        function block Node_F_VN_MaxElementElementwise_TcVnVector3_REAL [ST]: FB_init, Clone, OnExecute, PreExecutionCheck
        function block Node_F_VN_MaxElementElementwise_TcVnVector3_SINT [ST]: FB_init, Clone, OnExecute, PreExecutionCheck
        function block Node_F_VN_MaxElementElementwise_TcVnVector3_UINT [ST]: FB_init, Clone, OnExecute, PreExecutionCheck
        function block Node_F_VN_MaxElementElementwise_TcVnVector3_USINT [ST]: FB_init, Clone, OnExecute, PreExecutionCheck
        function block Node_F_VN_MaxElementElementwise_TcVnVector4_DINT [ST]: FB_init, Clone, OnExecute, PreExecutionCheck
        function block Node_F_VN_MaxElementElementwise_TcVnVector4_INT [ST]: FB_init, Clone, OnExecute, PreExecutionCheck
        function block Node_F_VN_MaxElementElementwise_TcVnVector4_LREAL [ST]: FB_init, Clone, OnExecute, PreExecutionCheck
        function block Node_F_VN_MaxElementElementwise_TcVnVector4_REAL [ST]: FB_init, Clone, OnExecute, PreExecutionCheck
        function block Node_F_VN_MaxElementElementwise_TcVnVector4_SINT [ST]: FB_init, Clone, OnExecute, PreExecutionCheck
        function block Node_F_VN_MaxElementElementwise_TcVnVector4_UINT [ST]: FB_init, Clone, OnExecute, PreExecutionCheck
        function block Node_F_VN_MaxElementElementwise_TcVnVector4_USINT [ST]: FB_init, Clone, OnExecute, PreExecutionCheck
        function block Node_F_VN_MaxElementElementwise_UDINT [ST]: FB_init, Clone, OnExecute, PreExecutionCheck
        function block Node_F_VN_MaxElementElementwise_UINT [ST]: FB_init, Clone, OnExecute, PreExecutionCheck
        function block Node_F_VN_MaxElementElementwise_ULINT [ST]: FB_init, Clone, OnExecute, PreExecutionCheck
        function block Node_F_VN_MaxElementElementwise_USINT [ST]: FB_init, Clone, OnExecute, PreExecutionCheck
      MedianElementwise/
        function block Node_F_VN_MedianElementElementwise_DINT [ST]: FB_init, Clone, OnExecute, PreExecutionCheck
        function block Node_F_VN_MedianElementElementwise_INT [ST]: FB_init, Clone, OnExecute, PreExecutionCheck
        function block Node_F_VN_MedianElementElementwise_LREAL [ST]: FB_init, Clone, OnExecute, PreExecutionCheck
        function block Node_F_VN_MedianElementElementwise_REAL [ST]: FB_init, Clone, OnExecute, PreExecutionCheck
        function block Node_F_VN_MedianElementElementwise_SINT [ST]: FB_init, Clone, OnExecute, PreExecutionCheck
        function block Node_F_VN_MedianElementElementwise_TcVnPoint2_DINT [ST]: FB_init, Clone, OnExecute, PreExecutionCheck
        function block Node_F_VN_MedianElementElementwise_TcVnPoint2_LREAL [ST]: FB_init, Clone, OnExecute, PreExecutionCheck
        function block Node_F_VN_MedianElementElementwise_TcVnPoint2_REAL [ST]: FB_init, Clone, OnExecute, PreExecutionCheck
        function block Node_F_VN_MedianElementElementwise_TcVnPoint3_LREAL [ST]: FB_init, Clone, OnExecute, PreExecutionCheck
        function block Node_F_VN_MedianElementElementwise_TcVnPoint3_REAL [ST]: FB_init, Clone, OnExecute, PreExecutionCheck
        function block Node_F_VN_MedianElementElementwise_TcVnVector2_DINT [ST]: FB_init, Clone, OnExecute, PreExecutionCheck
        function block Node_F_VN_MedianElementElementwise_TcVnVector2_INT [ST]: FB_init, Clone, OnExecute, PreExecutionCheck
        function block Node_F_VN_MedianElementElementwise_TcVnVector2_REAL [ST]: FB_init, Clone, OnExecute, PreExecutionCheck
        function block Node_F_VN_MedianElementElementwise_TcVnVector2_SINT [ST]: FB_init, Clone, OnExecute, PreExecutionCheck
        function block Node_F_VN_MedianElementElementwise_TcVnVector2_UINT [ST]: FB_init, Clone, OnExecute, PreExecutionCheck
        function block Node_F_VN_MedianElementElementwise_TcVnVector2_USINT [ST]: FB_init, Clone, OnExecute, PreExecutionCheck
        function block Node_F_VN_MedianElementElementwise_TcVnVector3_INT [ST]: FB_init, Clone, OnExecute, PreExecutionCheck
        function block Node_F_VN_MedianElementElementwise_TcVnVector3_REAL [ST]: FB_init, Clone, OnExecute, PreExecutionCheck
        function block Node_F_VN_MedianElementElementwise_TcVnVector3_SINT [ST]: FB_init, Clone, OnExecute, PreExecutionCheck
        function block Node_F_VN_MedianElementElementwise_TcVnVector3_UINT [ST]: FB_init, Clone, OnExecute, PreExecutionCheck
        function block Node_F_VN_MedianElementElementwise_TcVnVector3_USINT [ST]: FB_init, Clone, OnExecute, PreExecutionCheck
        function block Node_F_VN_MedianElementElementwise_TcVnVector4_DINT [ST]: FB_init, Clone, OnExecute, PreExecutionCheck
        function block Node_F_VN_MedianElementElementwise_TcVnVector4_INT [ST]: FB_init, Clone, OnExecute, PreExecutionCheck
        function block Node_F_VN_MedianElementElementwise_TcVnVector4_LREAL [ST]: FB_init, Clone, OnExecute, PreExecutionCheck
        function block Node_F_VN_MedianElementElementwise_TcVnVector4_REAL [ST]: FB_init, Clone, OnExecute, PreExecutionCheck
        function block Node_F_VN_MedianElementElementwise_TcVnVector4_SINT [ST]: FB_init, Clone, OnExecute, PreExecutionCheck
        function block Node_F_VN_MedianElementElementwise_TcVnVector4_UINT [ST]: FB_init, Clone, OnExecute, PreExecutionCheck
        function block Node_F_VN_MedianElementElementwise_TcVnVector4_USINT [ST]: FB_init, Clone, OnExecute, PreExecutionCheck
        function block Node_F_VN_MedianElementElementwise_UDINT [ST]: FB_init, Clone, OnExecute, PreExecutionCheck
        function block Node_F_VN_MedianElementElementwise_UINT [ST]: FB_init, Clone, OnExecute, PreExecutionCheck
        function block Node_F_VN_MedianElementElementwise_ULINT [ST]: FB_init, Clone, OnExecute, PreExecutionCheck
        function block Node_F_VN_MedianElementElementwise_USINT [ST]: FB_init, Clone, OnExecute, PreExecutionCheck
      MinElementwise/
        function block Node_F_VN_MinElementElementwise_DINT [ST]: FB_init, Clone, OnExecute, PreExecutionCheck
        function block Node_F_VN_MinElementElementwise_INT [ST]: FB_init, Clone, OnExecute, PreExecutionCheck
        function block Node_F_VN_MinElementElementwise_LREAL [ST]: FB_init, Clone, OnExecute, PreExecutionCheck
        function block Node_F_VN_MinElementElementwise_REAL [ST]: FB_init, Clone, OnExecute, PreExecutionCheck
        function block Node_F_VN_MinElementElementwise_SINT [ST]: FB_init, Clone, OnExecute, PreExecutionCheck
        function block Node_F_VN_MinElementElementwise_TcVnPoint2_DINT [ST]: FB_init, Clone, OnExecute, PreExecutionCheck
        function block Node_F_VN_MinElementElementwise_TcVnPoint2_LREAL [ST]: FB_init, Clone, OnExecute, PreExecutionCheck
        function block Node_F_VN_MinElementElementwise_TcVnPoint2_REAL [ST]: FB_init, Clone, OnExecute, PreExecutionCheck
        function block Node_F_VN_MinElementElementwise_TcVnPoint3_LREAL [ST]: FB_init, Clone, OnExecute, PreExecutionCheck
        function block Node_F_VN_MinElementElementwise_TcVnPoint3_REAL [ST]: FB_init, Clone, OnExecute, PreExecutionCheck
        function block Node_F_VN_MinElementElementwise_TcVnVector2_DINT [ST]: FB_init, Clone, OnExecute, PreExecutionCheck
        function block Node_F_VN_MinElementElementwise_TcVnVector2_INT [ST]: FB_init, Clone, OnExecute, PreExecutionCheck
        function block Node_F_VN_MinElementElementwise_TcVnVector2_REAL [ST]: FB_init, Clone, OnExecute, PreExecutionCheck
        function block Node_F_VN_MinElementElementwise_TcVnVector2_SINT [ST]: FB_init, Clone, OnExecute, PreExecutionCheck
        function block Node_F_VN_MinElementElementwise_TcVnVector2_UINT [ST]: FB_init, Clone, OnExecute, PreExecutionCheck
        function block Node_F_VN_MinElementElementwise_TcVnVector2_USINT [ST]: FB_init, Clone, OnExecute, PreExecutionCheck
        function block Node_F_VN_MinElementElementwise_TcVnVector3_INT [ST]: FB_init, Clone, OnExecute, PreExecutionCheck
        function block Node_F_VN_MinElementElementwise_TcVnVector3_REAL [ST]: FB_init, Clone, OnExecute, PreExecutionCheck
        function block Node_F_VN_MinElementElementwise_TcVnVector3_SINT [ST]: FB_init, Clone, OnExecute, PreExecutionCheck
        function block Node_F_VN_MinElementElementwise_TcVnVector3_UINT [ST]: FB_init, Clone, OnExecute, PreExecutionCheck
        function block Node_F_VN_MinElementElementwise_TcVnVector3_USINT [ST]: FB_init, Clone, OnExecute, PreExecutionCheck
        function block Node_F_VN_MinElementElementwise_TcVnVector4_DINT [ST]: FB_init, Clone, OnExecute, PreExecutionCheck
        function block Node_F_VN_MinElementElementwise_TcVnVector4_INT [ST]: FB_init, Clone, OnExecute, PreExecutionCheck
        function block Node_F_VN_MinElementElementwise_TcVnVector4_LREAL [ST]: FB_init, Clone, OnExecute, PreExecutionCheck
        function block Node_F_VN_MinElementElementwise_TcVnVector4_REAL [ST]: FB_init, Clone, OnExecute, PreExecutionCheck
        function block Node_F_VN_MinElementElementwise_TcVnVector4_SINT [ST]: FB_init, Clone, OnExecute, PreExecutionCheck
        function block Node_F_VN_MinElementElementwise_TcVnVector4_UINT [ST]: FB_init, Clone, OnExecute, PreExecutionCheck
        function block Node_F_VN_MinElementElementwise_TcVnVector4_USINT [ST]: FB_init, Clone, OnExecute, PreExecutionCheck
        function block Node_F_VN_MinElementElementwise_UDINT [ST]: FB_init, Clone, OnExecute, PreExecutionCheck
        function block Node_F_VN_MinElementElementwise_UINT [ST]: FB_init, Clone, OnExecute, PreExecutionCheck
        function block Node_F_VN_MinElementElementwise_ULINT [ST]: FB_init, Clone, OnExecute, PreExecutionCheck
        function block Node_F_VN_MinElementElementwise_USINT [ST]: FB_init, Clone, OnExecute, PreExecutionCheck
      function block Node_F_VN_ContainerAverage [ST]: FB_init, Clone, OnExecute, PreExecutionCheck
      function block Node_F_VN_ContainerAverageElementwise2 [ST]: FB_init, Clone, OnExecute, PreExecutionCheck
      function block Node_F_VN_ContainerAverageElementwise3 [ST]: FB_init, Clone, OnExecute, PreExecutionCheck
      function block Node_F_VN_ContainerAverageElementwise4 [ST]: FB_init, Clone, OnExecute, PreExecutionCheck
      function block Node_F_VN_ContainerAverageVariance [ST]: FB_init, Clone, OnExecute, PreExecutionCheck
      function block Node_F_VN_ContainerAverageVarianceElementwise2 [ST]: FB_init, Clone, OnExecute, PreExecutionCheck
      function block Node_F_VN_ContainerAverageVarianceElementwise3 [ST]: FB_init, Clone, OnExecute, PreExecutionCheck
      function block Node_F_VN_ContainerAverageVarianceElementwise4 [ST]: FB_init, Clone, OnExecute, PreExecutionCheck
      function block Node_F_VN_MaxElement [ST]: FB_init, Clone, OnExecute, PreExecutionCheck
      function block Node_F_VN_MedianElement [ST]: FB_init, Clone, OnExecute, PreExecutionCheck
      function block Node_F_VN_MinElement [ST]: FB_init, Clone, OnExecute, PreExecutionCheck
    Contour Analysis/
      function block Node_F_VN_ApproximatePolygon [ST]: FB_init, Clone, OnExecute, PreExecutionCheck
      function block Node_F_VN_CheckIfPointIsInsideContour [ST]: FB_init, Clone, OnExecute, PreExecutionCheck
      function block Node_F_VN_ContourArea [ST]: FB_init, Clone, OnExecute, PreExecutionCheck
      function block Node_F_VN_ContourCenterOfMass [ST]: FB_init, Clone, OnExecute, PreExecutionCheck
      function block Node_F_VN_ContourCircularity [ST]: FB_init, Clone, OnExecute, PreExecutionCheck
      function block Node_F_VN_ContourCircularityExp [ST]: FB_init, Clone, OnExecute, PreExecutionCheck
      function block Node_F_VN_ContourConvexity [ST]: FB_init, Clone, OnExecute, PreExecutionCheck
      function block Node_F_VN_ContourEccentricity [ST]: FB_init, Clone, OnExecute, PreExecutionCheck
      function block Node_F_VN_ContourElongation [ST]: FB_init, Clone, OnExecute, PreExecutionCheck
      function block Node_F_VN_ContourExtremePoint [ST]: FB_init, Clone, OnExecute, PreExecutionCheck
      function block Node_F_VN_ContourInertiaRatio [ST]: FB_init, Clone, OnExecute, PreExecutionCheck
      function block Node_F_VN_ContourMoments [ST]: FB_init, Clone, OnExecute, PreExecutionCheck
      function block Node_F_VN_ContourOrientation [ST]: FB_init, Clone, OnExecute, PreExecutionCheck
      function block Node_F_VN_ContourOrientationExp [ST]: FB_init, Clone, OnExecute, PreExecutionCheck
      function block Node_F_VN_ContourPerimeter [ST]: FB_init, Clone, OnExecute, PreExecutionCheck
      function block Node_F_VN_ContourRoundness [ST]: FB_init, Clone, OnExecute, PreExecutionCheck
      function block Node_F_VN_ConvexHullPoints [ST]: FB_init, Clone, OnExecute, PreExecutionCheck
      function block Node_F_VN_ConvexHullPointsExp [ST]: FB_init, Clone, OnExecute, PreExecutionCheck
      function block Node_F_VN_ConvexityDefects [ST]: FB_init, Clone, OnExecute, PreExecutionCheck
      function block Node_F_VN_EnclosingCircle [ST]: FB_init, Clone, OnExecute, PreExecutionCheck
      function block Node_F_VN_EnclosingRectangle [ST]: FB_init, Clone, OnExecute, PreExecutionCheck
      function block Node_F_VN_EnclosingTriangle [ST]: FB_init, Clone, OnExecute, PreExecutionCheck
      function block Node_F_VN_FitEllipse [ST]: FB_init, Clone, OnExecute, PreExecutionCheck
      function block Node_F_VN_FitLine [ST]: FB_init, Clone, OnExecute, PreExecutionCheck
      function block Node_F_VN_FitLineExp [ST]: FB_init, Clone, OnExecute, PreExecutionCheck
      function block Node_F_VN_MatchContours [ST]: FB_init, Clone, OnExecute, PreExecutionCheck
      function block Node_F_VN_MatchContours1vsN [ST]: FB_init, Clone, OnExecute, PreExecutionCheck
      function block Node_F_VN_MatchContours1vsNExp [ST]: FB_init, Clone, OnExecute, PreExecutionCheck
      function block Node_F_VN_MatchContoursExp [ST]: FB_init, Clone, OnExecute, PreExecutionCheck
      function block Node_F_VN_UprightBoundingRectangle [ST]: FB_init, Clone, OnExecute, PreExecutionCheck
    Control Functions/
    Drawing/
      function block Node_F_VN_DrawArrow [ST]: FB_init, Clone, OnExecute, PreExecutionCheck
      function block Node_F_VN_DrawArrow_TcVnVector4_DINT [ST]: FB_init, Clone, OnExecute, PreExecutionCheck
      function block Node_F_VN_DrawArrowExp [ST]: FB_init, Clone, OnExecute, PreExecutionCheck
      function block Node_F_VN_DrawArrowExp_TcVnVector4_DINT [ST]: FB_init, Clone, OnExecute, PreExecutionCheck
      function block Node_F_VN_DrawCircle [ST]: FB_init, Clone, OnExecute, PreExecutionCheck
      function block Node_F_VN_DrawCircleExp [ST]: FB_init, Clone, OnExecute, PreExecutionCheck
      function block Node_F_VN_DrawCircles [ST]: FB_init, Clone, OnExecute, PreExecutionCheck
      function block Node_F_VN_DrawCirclesExp [ST]: FB_init, Clone, OnExecute, PreExecutionCheck
      function block Node_F_VN_DrawCircularArc [ST]: FB_init, Clone, OnExecute, PreExecutionCheck
      function block Node_F_VN_DrawCircularArcExp [ST]: FB_init, Clone, OnExecute, PreExecutionCheck
      function block Node_F_VN_DrawComponents [ST]: FB_init, Clone, OnExecute, PreExecutionCheck
      function block Node_F_VN_DrawComponentsExp [ST]: FB_init, Clone, OnExecute, PreExecutionCheck
      function block Node_F_VN_DrawContours [ST]: FB_init, Clone, OnExecute, PreExecutionCheck
      function block Node_F_VN_DrawContoursExp [ST]: FB_init, Clone, OnExecute, PreExecutionCheck
      function block Node_F_VN_DrawEllipse [ST]: FB_init, Clone, OnExecute, PreExecutionCheck
      function block Node_F_VN_DrawEllipseExp [ST]: FB_init, Clone, OnExecute, PreExecutionCheck
      function block Node_F_VN_DrawKeypoints [ST]: FB_init, Clone, OnExecute, PreExecutionCheck
      function block Node_F_VN_DrawKeypointsExp [ST]: FB_init, Clone, OnExecute, PreExecutionCheck
      function block Node_F_VN_DrawLine [ST]: FB_init, Clone, OnExecute, PreExecutionCheck
      function block Node_F_VN_DrawLine_TcVnVector4_DINT [ST]: FB_init, Clone, OnExecute, PreExecutionCheck
      function block Node_F_VN_DrawLine_TcVnVector4_LREAL [ST]: FB_init, Clone, OnExecute, PreExecutionCheck
      function block Node_F_VN_DrawLineExp [ST]: FB_init, Clone, OnExecute, PreExecutionCheck
      function block Node_F_VN_DrawLineExp_TcVnVector4_DINT [ST]: FB_init, Clone, OnExecute, PreExecutionCheck
      function block Node_F_VN_DrawLineExp_TcVnVector4_LREAL [ST]: FB_init, Clone, OnExecute, PreExecutionCheck
      function block Node_F_VN_DrawLines [ST]: FB_init, Clone, OnExecute, PreExecutionCheck
      function block Node_F_VN_DrawLinesExp [ST]: FB_init, Clone, OnExecute, PreExecutionCheck
      function block Node_F_VN_DrawMatches [ST]: FB_init, Clone, OnExecute, PreExecutionCheck
      function block Node_F_VN_DrawMatchesExp [ST]: FB_init, Clone, OnExecute, PreExecutionCheck
      function block Node_F_VN_DrawOrientation [ST]: FB_init, Clone, OnExecute, PreExecutionCheck
      function block Node_F_VN_DrawOrientationExp [ST]: FB_init, Clone, OnExecute, PreExecutionCheck
      function block Node_F_VN_DrawPoint [ST]: FB_init, Clone, OnExecute, PreExecutionCheck
      function block Node_F_VN_DrawPointExp [ST]: FB_init, Clone, OnExecute, PreExecutionCheck
      function block Node_F_VN_DrawPoints [ST]: FB_init, Clone, OnExecute, PreExecutionCheck
      function block Node_F_VN_DrawPointsExp [ST]: FB_init, Clone, OnExecute, PreExecutionCheck
      function block Node_F_VN_DrawPolygon [ST]: FB_init, Clone, OnExecute, PreExecutionCheck
      function block Node_F_VN_DrawPolygonExp [ST]: FB_init, Clone, OnExecute, PreExecutionCheck
      function block Node_F_VN_DrawRectangle [ST]: FB_init, Clone, OnExecute, PreExecutionCheck
      function block Node_F_VN_DrawRectangle_TcVnRectangle_DINT [ST]: FB_init, Clone, OnExecute, PreExecutionCheck
      function block Node_F_VN_DrawRectangle_TcVnRectangle_UDINT [ST]: FB_init, Clone, OnExecute, PreExecutionCheck
      function block Node_F_VN_DrawRotatedRectangle [ST]: FB_init, Clone, OnExecute, PreExecutionCheck
      function block Node_F_VN_DrawRotatedRectangleExp [ST]: FB_init, Clone, OnExecute, PreExecutionCheck
      function block Node_F_VN_FillCircle [ST]: FB_init, Clone, OnExecute, PreExecutionCheck
      function block Node_F_VN_FillContours [ST]: FB_init, Clone, OnExecute, PreExecutionCheck
      function block Node_F_VN_FillEllipse [ST]: FB_init, Clone, OnExecute, PreExecutionCheck
      function block Node_F_VN_FillPolygon [ST]: FB_init, Clone, OnExecute, PreExecutionCheck
      function block Node_F_VN_FillRectangle [ST]: FB_init, Clone, OnExecute, PreExecutionCheck
      function block Node_F_VN_FillRotatedRectangle [ST]: FB_init, Clone, OnExecute, PreExecutionCheck
      function block Node_F_VN_PlotIntensityProfile [ST]: FB_init, Clone, OnExecute, PreExecutionCheck
      function block Node_F_VN_PlotIntensityProfileExp [ST]: FB_init, Clone, OnExecute, PreExecutionCheck
      function block Node_F_VN_PutLabel [ST]: FB_init, Clone, OnExecute, PreExecutionCheck
      function block Node_F_VN_PutLabelExp [ST]: FB_init, Clone, OnExecute, PreExecutionCheck
      function block Node_F_VN_PutText [ST]: FB_init, Clone, OnExecute, PreExecutionCheck
      function block Node_F_VN_PutTextExp [ST]: FB_init, Clone, OnExecute, PreExecutionCheck
    Fourier Analysis/
      function block Node_F_VN_CreateBandpassButterworthFilter [ST]: FB_init, Clone, OnExecute, PreExecutionCheck
      function block Node_F_VN_CreateBandpassGaussianFilter [ST]: FB_init, Clone, OnExecute, PreExecutionCheck
      function block Node_F_VN_CreateBandrejectButterworthFilter [ST]: FB_init, Clone, OnExecute, PreExecutionCheck
      function block Node_F_VN_CreateBandrejectGaussianFilter [ST]: FB_init, Clone, OnExecute, PreExecutionCheck
      function block Node_F_VN_CreateHighpassButterworthFilter [ST]: FB_init, Clone, OnExecute, PreExecutionCheck
      function block Node_F_VN_CreateHighpassGaussianFilter [ST]: FB_init, Clone, OnExecute, PreExecutionCheck
      function block Node_F_VN_CreateLowpassButterworthFilter [ST]: FB_init, Clone, OnExecute, PreExecutionCheck
      function block Node_F_VN_CreateLowpassGaussianFilter [ST]: FB_init, Clone, OnExecute, PreExecutionCheck
      function block Node_F_VN_Dft [ST]: FB_init, Clone, OnExecute, PreExecutionCheck
      function block Node_F_VN_InverseDft [ST]: FB_init, Clone, OnExecute, PreExecutionCheck
      function block Node_F_VN_OptimalDftSize [ST]: FB_init, Clone, OnExecute, PreExecutionCheck
    Geometric and Coord Transform/
      Calibration/
        function block Node_F_VN_CalibrateCamera [ST]: FB_init, Clone, OnExecute, PreExecutionCheck
        function block Node_F_VN_CalibrateCameraPlanar [ST]: FB_init, Clone, OnExecute, PreExecutionCheck
        function block Node_F_VN_CompensateLensDistortion [ST]: FB_init, Clone, OnExecute, PreExecutionCheck
        function block Node_F_VN_CompensateLensDistortionExp1 [ST]: FB_init, Clone, OnExecute, PreExecutionCheck
        function block Node_F_VN_CompensateLensDistortionExp2 [ST]: FB_init, Clone, OnExecute, PreExecutionCheck
        function block Node_F_VN_CompensateLensDistortionForPoints [ST]: FB_init, Clone, OnExecute, PreExecutionCheck
        function block Node_F_VN_CompensateLensDistortionForPointsExp1 [ST]: FB_init, Clone, OnExecute, PreExecutionCheck
        function block Node_F_VN_CompensateLensDistortionForPointsExp2 [ST]: FB_init, Clone, OnExecute, PreExecutionCheck
        function block Node_F_VN_DetectPatternPoints [ST]: FB_init, Clone, OnExecute, PreExecutionCheck
        function block Node_F_VN_GenerateCalibrationPatternReferencePoints [ST]: FB_init, Clone, OnExecute, PreExecutionCheck
        function block Node_F_VN_SolvePnP [ST]: FB_init, Clone, OnExecute, PreExecutionCheck
        function block Node_F_VN_SolvePnPExp [ST]: FB_init, Clone, OnExecute, PreExecutionCheck
        function block Node_F_VN_SortDetectedPatternPoints [ST]: FB_init, Clone, OnExecute, PreExecutionCheck
      function block Node_F_VN_AlignRotatedImageRegion [ST]: FB_init, Clone, OnExecute, PreExecutionCheck
      function block Node_F_VN_AlignRotatedImageRegionExp [ST]: FB_init, Clone, OnExecute, PreExecutionCheck
      function block Node_F_VN_ApplyRotationToAffineTransformation [ST]: FB_init, Clone, OnExecute, PreExecutionCheck
      function block Node_F_VN_ApplyRotationToAffineTransformationExp [ST]: FB_init, Clone, OnExecute, PreExecutionCheck
      function block Node_F_VN_ApplyScalingToAffineTransformation [ST]: FB_init, Clone, OnExecute, PreExecutionCheck
      function block Node_F_VN_ApplyScalingToAffineTransformationExp [ST]: FB_init, Clone, OnExecute, PreExecutionCheck
      function block Node_F_VN_ApplyTranslationToAffineTransformation [ST]: FB_init, Clone, OnExecute, PreExecutionCheck
      function block Node_F_VN_ApplyTranslationToAffineTransformationExp [ST]: FB_init, Clone, OnExecute, PreExecutionCheck
      function block Node_F_VN_ApplyYAxisInversionToAffineTransformation [ST]: FB_init, Clone, OnExecute, PreExecutionCheck
      function block Node_F_VN_ApplyYAxisInversionToAffineTransformationExp [ST]: FB_init, Clone, OnExecute, PreExecutionCheck
      function block Node_F_VN_ConvertCartesianToPolarAngleImage [ST]: FB_init, Clone, OnExecute, PreExecutionCheck
      function block Node_F_VN_ConvertCartesianToPolarAngleImageExp [ST]: FB_init, Clone, OnExecute, PreExecutionCheck
      function block Node_F_VN_ConvertCartesianToPolarAngles [ST]: FB_init, Clone, OnExecute, PreExecutionCheck
      function block Node_F_VN_ConvertCartesianToPolarAnglesExp [ST]: FB_init, Clone, OnExecute, PreExecutionCheck
      function block Node_F_VN_ConvertCartesianToPolarImages [ST]: FB_init, Clone, OnExecute, PreExecutionCheck
      function block Node_F_VN_ConvertCartesianToPolarImagesExp [ST]: FB_init, Clone, OnExecute, PreExecutionCheck
      function block Node_F_VN_ConvertCartesianToPolarMagnitudeImage [ST]: FB_init, Clone, OnExecute, PreExecutionCheck
      function block Node_F_VN_ConvertCartesianToPolarMagnitudes [ST]: FB_init, Clone, OnExecute, PreExecutionCheck
      function block Node_F_VN_ConvertCartesianToPolarPoints [ST]: FB_init, Clone, OnExecute, PreExecutionCheck
      function block Node_F_VN_ConvertCartesianToPolarPointsExp [ST]: FB_init, Clone, OnExecute, PreExecutionCheck
      function block Node_F_VN_ConvertMaps [ST]: FB_init, Clone, OnExecute, PreExecutionCheck
      function block Node_F_VN_ConvertPolarToCartesianImages [ST]: FB_init, Clone, OnExecute, PreExecutionCheck
      function block Node_F_VN_ConvertPolarToCartesianImagesExp [ST]: FB_init, Clone, OnExecute, PreExecutionCheck
      function block Node_F_VN_ConvertPolarToCartesianPoints [ST]: FB_init, Clone, OnExecute, PreExecutionCheck
      function block Node_F_VN_ConvertPolarToCartesianPointsExp [ST]: FB_init, Clone, OnExecute, PreExecutionCheck
      function block Node_F_VN_DecomposeAffineTransformation [ST]: FB_init, Clone, OnExecute, PreExecutionCheck
      function block Node_F_VN_DecomposeAffineTransformationExp [ST]: FB_init, Clone, OnExecute, PreExecutionCheck
      function block Node_F_VN_FlipImage [ST]: FB_init, Clone, OnExecute, PreExecutionCheck
      function block Node_F_VN_GenerateAffineTransformationUnitMatrix2D [ST]: FB_init, Clone, OnExecute, PreExecutionCheck
      function block Node_F_VN_GetAffineTransformation [ST]: FB_init, Clone, OnExecute, PreExecutionCheck
      function block Node_F_VN_GetAffineTransformation2D [ST]: FB_init, Clone, OnExecute, PreExecutionCheck
      function block Node_F_VN_GetPerspectiveTransformation [ST]: FB_init, Clone, OnExecute, PreExecutionCheck
      function block Node_F_VN_Homography [ST]: FB_init, Clone, OnExecute, PreExecutionCheck
      function block Node_F_VN_HomographyExp [ST]: FB_init, Clone, OnExecute, PreExecutionCheck
      function block Node_F_VN_InvertAffineTransformation [ST]: FB_init, Clone, OnExecute, PreExecutionCheck
      function block Node_F_VN_PerspectiveTransformation [ST]: FB_init, Clone, OnExecute, PreExecutionCheck
      function block Node_F_VN_PyramidDown [ST]: FB_init, Clone, OnExecute, PreExecutionCheck
      function block Node_F_VN_PyramidUp [ST]: FB_init, Clone, OnExecute, PreExecutionCheck
      function block Node_F_VN_RemapImage [ST]: FB_init, Clone, OnExecute, PreExecutionCheck
      function block Node_F_VN_RemapImageExp [ST]: FB_init, Clone, OnExecute, PreExecutionCheck
      function block Node_F_VN_RemapImageToLogPolarSpace [ST]: FB_init, Clone, OnExecute, PreExecutionCheck
      function block Node_F_VN_RemapImageToLogPolarSpaceExp [ST]: FB_init, Clone, OnExecute, PreExecutionCheck
      function block Node_F_VN_RemapImageToLogPolarSpaceExp2 [ST]: FB_init, Clone, OnExecute, PreExecutionCheck
      function block Node_F_VN_RemapImageToPolarSpace [ST]: FB_init, Clone, OnExecute, PreExecutionCheck
      function block Node_F_VN_RemapImageToPolarSpaceExp [ST]: FB_init, Clone, OnExecute, PreExecutionCheck
      function block Node_F_VN_RemapImageToPolarSpaceExp2 [ST]: FB_init, Clone, OnExecute, PreExecutionCheck
      function block Node_F_VN_ResizeImage [ST]: FB_init, Clone, OnExecute, PreExecutionCheck
      function block Node_F_VN_ResizeImageExp [ST]: FB_init, Clone, OnExecute, PreExecutionCheck
      function block Node_F_VN_ResizeRegion_TcVnRectangle_DINT [ST]: FB_init, Clone, OnExecute, PreExecutionCheck
      function block Node_F_VN_RotateImage [ST]: FB_init, Clone, OnExecute, PreExecutionCheck
      function block Node_F_VN_RotateImageExp [ST]: FB_init, Clone, OnExecute, PreExecutionCheck
      function block Node_F_VN_RotateImageExp2 [ST]: FB_init, Clone, OnExecute, PreExecutionCheck
      function block Node_F_VN_WarpAffine [ST]: FB_init, Clone, OnExecute, PreExecutionCheck
      function block Node_F_VN_WarpAffine_Container [ST]: FB_init, Clone, OnExecute, PreExecutionCheck
      function block Node_F_VN_WarpAffine_Point [ST]: FB_init, Clone, OnExecute, PreExecutionCheck
      function block Node_F_VN_WarpAffine_Rectangle [ST]: FB_init, Clone, OnExecute, PreExecutionCheck
      function block Node_F_VN_WarpAffineExp [ST]: FB_init, Clone, OnExecute, PreExecutionCheck
      function block Node_F_VN_WarpPerspective [ST]: FB_init, Clone, OnExecute, PreExecutionCheck
      function block Node_F_VN_WarpPerspective_Container [ST]: FB_init, Clone, OnExecute, PreExecutionCheck
      function block Node_F_VN_WarpPerspective_Point [ST]: FB_init, Clone, OnExecute, PreExecutionCheck
      function block Node_F_VN_WarpPerspective_Rectangle [ST]: FB_init, Clone, OnExecute, PreExecutionCheck
      function block Node_F_VN_WarpPerspectiveExp [ST]: FB_init, Clone, OnExecute, PreExecutionCheck
    Helpers/
      function block Node_Mux10Way_ITcVnImage [ST]: FB_init, Clone, OnExecute
    Image Analysis/
      Object Detection/
        function block Node_F_VN_DetectBlobs [ST]: FB_init, Clone, OnExecute, PreExecutionCheck
        function block Node_F_VN_DetectBlobsExp [ST]: FB_init, Clone, OnExecute, PreExecutionCheck
        function block Node_F_VN_FindContourHierarchyExp [ST]: FB_init, Clone, OnExecute, PreExecutionCheck
        function block Node_F_VN_FindContours [ST]: FB_init, Clone, OnExecute, PreExecutionCheck
        function block Node_F_VN_FindContoursExp [ST]: FB_init, Clone, OnExecute, PreExecutionCheck
        function block Node_F_VN_FindRois [ST]: FB_init, Clone, OnExecute, PreExecutionCheck
        function block Node_F_VN_FindTemplateWalsh [ST]: FB_init, Clone, OnExecute, PreExecutionCheck
        function block Node_F_VN_FindTemplateWalsh_AngleRange [ST]: FB_init, Clone, OnExecute, PreExecutionCheck
        function block Node_F_VN_FindTemplateWalshExp [ST]: FB_init, Clone, OnExecute, PreExecutionCheck
        function block Node_F_VN_FindTemplateWalshExp_AngleRange [ST]: FB_init, Clone, OnExecute, PreExecutionCheck
        function block Node_F_VN_HoughCircles [ST]: FB_init, Clone, OnExecute, PreExecutionCheck
        function block Node_F_VN_HoughCirclesExp [ST]: FB_init, Clone, OnExecute, PreExecutionCheck
        function block Node_F_VN_HoughLines [ST]: FB_init, Clone, OnExecute, PreExecutionCheck
        function block Node_F_VN_HoughLinesP [ST]: FB_init, Clone, OnExecute, PreExecutionCheck
        function block Node_F_VN_HoughLinesPExp [ST]: FB_init, Clone, OnExecute, PreExecutionCheck
        function block Node_F_VN_MatchImageHuMoments [ST]: FB_init, Clone, OnExecute, PreExecutionCheck
        function block Node_F_VN_MatchTemplate [ST]: FB_init, Clone, OnExecute, PreExecutionCheck
        function block Node_F_VN_MatchTemplateAndEvaluate [ST]: FB_init, Clone, OnExecute, PreExecutionCheck
        function block Node_F_VN_MatchTemplateAndEvaluateExp [ST]: FB_init, Clone, OnExecute, PreExecutionCheck
        function block Node_F_VN_MatchTemplateExp [ST]: FB_init, Clone, OnExecute, PreExecutionCheck
        function block Node_F_VN_MatchTemplateWalsh [ST]: FB_init, Clone, OnExecute, PreExecutionCheck
        function block Node_F_VN_MatchTemplateWalshExp [ST]: FB_init, Clone, OnExecute, PreExecutionCheck
        function block Node_F_VN_MergeRegions [ST]: FB_init, Clone, OnExecute, PreExecutionCheck
        function block Node_F_VN_SalientFeatures [ST]: FB_init, Clone, OnExecute, PreExecutionCheck
      function block Node_F_VN_CannyEdgeDetection [ST]: FB_init, Clone, OnExecute, PreExecutionCheck
      function block Node_F_VN_CannyEdgeDetectionExp [ST]: FB_init, Clone, OnExecute, PreExecutionCheck
      function block Node_F_VN_ConnectedComponents [ST]: FB_init, Clone, OnExecute, PreExecutionCheck
      function block Node_F_VN_ConnectedComponentsExp [ST]: FB_init, Clone, OnExecute, PreExecutionCheck
      function block Node_F_VN_ConnectedComponentsWithStats [ST]: FB_init, Clone, OnExecute, PreExecutionCheck
      function block Node_F_VN_ConnectedComponentsWithStatsExp [ST]: FB_init, Clone, OnExecute, PreExecutionCheck
      function block Node_F_VN_CountNonZeroPixels [ST]: FB_init, Clone, OnExecute, PreExecutionCheck
      function block Node_F_VN_DistanceTransformation [ST]: FB_init, Clone, OnExecute, PreExecutionCheck
      function block Node_F_VN_DistanceTransformationExp [ST]: FB_init, Clone, OnExecute, PreExecutionCheck
      function block Node_F_VN_GetConnectedComponent [ST]: FB_init, Clone, OnExecute, PreExecutionCheck
      function block Node_F_VN_GetConnectedComponentExp [ST]: FB_init, Clone, OnExecute, PreExecutionCheck
      function block Node_F_VN_ImageAbsoluteAverage [ST]: FB_init, Clone, OnExecute, PreExecutionCheck
      function block Node_F_VN_ImageAverage [ST]: FB_init, Clone, OnExecute, PreExecutionCheck
      function block Node_F_VN_ImageAverageExp [ST]: FB_init, Clone, OnExecute, PreExecutionCheck
      function block Node_F_VN_ImageAverageStdDev [ST]: FB_init, Clone, OnExecute, PreExecutionCheck
      function block Node_F_VN_ImageAverageStdDevExp [ST]: FB_init, Clone, OnExecute, PreExecutionCheck
      function block Node_F_VN_ImageCenterOfMass [ST]: FB_init, Clone, OnExecute, PreExecutionCheck
      function block Node_F_VN_ImageCenterOfMassExp [ST]: FB_init, Clone, OnExecute, PreExecutionCheck
      function block Node_F_VN_ImageMedian [ST]: FB_init, Clone, OnExecute, PreExecutionCheck
      function block Node_F_VN_ImageMedianExp [ST]: FB_init, Clone, OnExecute, PreExecutionCheck
      function block Node_F_VN_ImageMoments [ST]: FB_init, Clone, OnExecute, PreExecutionCheck
      function block Node_F_VN_MaxPixelValue [ST]: FB_init, Clone, OnExecute, PreExecutionCheck
      function block Node_F_VN_MaxPixelValueExp [ST]: FB_init, Clone, OnExecute, PreExecutionCheck
      function block Node_F_VN_MinPixelValue [ST]: FB_init, Clone, OnExecute, PreExecutionCheck
      function block Node_F_VN_MinPixelValueExp [ST]: FB_init, Clone, OnExecute, PreExecutionCheck
      function block Node_F_VN_RegionOrientation [ST]: FB_init, Clone, OnExecute, PreExecutionCheck
      function block Node_F_VN_RegionOrientationExp [ST]: FB_init, Clone, OnExecute, PreExecutionCheck
      function block Node_F_VN_UprightInnerRectangle [ST]: FB_init, Clone, OnExecute, PreExecutionCheck
      function block Node_F_VN_UprightInnerRectangleExp [ST]: FB_init, Clone, OnExecute, PreExecutionCheck
    Image Color and Contrast Processing/
      function block Node_F_VN_ApplyColorMap [ST]: FB_init, Clone, OnExecute, PreExecutionCheck
      function block Node_F_VN_Clahe [ST]: FB_init, Clone, OnExecute, PreExecutionCheck
      function block Node_F_VN_ClaheExp [ST]: FB_init, Clone, OnExecute, PreExecutionCheck
      function block Node_F_VN_ConvertColorSpace [ST]: FB_init, Clone, OnExecute, PreExecutionCheck
      function block Node_F_VN_GenerateColorMap [ST]: FB_init, Clone, OnExecute, PreExecutionCheck
      function block Node_F_VN_GenerateCustomColorMap [ST]: FB_init, Clone, OnExecute, PreExecutionCheck
      function block Node_F_VN_Histogram [ST]: FB_init, Clone, OnExecute, PreExecutionCheck
      function block Node_F_VN_HistogramEqualization [ST]: FB_init, Clone, OnExecute, PreExecutionCheck
      function block Node_F_VN_HistogramEqualizationExp [ST]: FB_init, Clone, OnExecute, PreExecutionCheck
      function block Node_F_VN_HistogramExp [ST]: FB_init, Clone, OnExecute, PreExecutionCheck
      function block Node_F_VN_InvertImageColor [ST]: FB_init, Clone, OnExecute, PreExecutionCheck
      function block Node_F_VN_InvertImageColorExp [ST]: FB_init, Clone, OnExecute, PreExecutionCheck
      function block Node_F_VN_NormalizeImage [ST]: FB_init, Clone, OnExecute, PreExecutionCheck
      function block Node_F_VN_NormalizeImageExp [ST]: FB_init, Clone, OnExecute, PreExecutionCheck
      function block Node_F_VN_NormalizeImageForDisplay [ST]: FB_init, Clone, OnExecute, PreExecutionCheck
      function block Node_F_VN_ReferenceColorSimilarity_TcVnVector3_LREAL [ST]: FB_init, Clone, OnExecute, PreExecutionCheck
      function block Node_F_VN_ReferenceColorSimilarityExp_TcVnVector3_LREAL [ST]: FB_init, Clone, OnExecute, PreExecutionCheck
      function block Node_F_VN_WhiteBalance [ST]: FB_init, Clone, OnExecute, PreExecutionCheck
    Image Filtering/
      function block Node_F_VN_BilateralFilter [ST]: FB_init, Clone, OnExecute, PreExecutionCheck
      function block Node_F_VN_BilateralFilterExp [ST]: FB_init, Clone, OnExecute, PreExecutionCheck
      function block Node_F_VN_BoxFilter [ST]: FB_init, Clone, OnExecute, PreExecutionCheck
      function block Node_F_VN_BoxFilterExp [ST]: FB_init, Clone, OnExecute, PreExecutionCheck
      function block Node_F_VN_BrightBorderObjects [ST]: FB_init, Clone, OnExecute, PreExecutionCheck
      function block Node_F_VN_CreateStructuringElement [ST]: FB_init, Clone, OnExecute, PreExecutionCheck
      function block Node_F_VN_DarkBorderObjects [ST]: FB_init, Clone, OnExecute, PreExecutionCheck
      function block Node_F_VN_FillHoles [ST]: FB_init, Clone, OnExecute, PreExecutionCheck
      function block Node_F_VN_GaussianFilter [ST]: FB_init, Clone, OnExecute, PreExecutionCheck
      function block Node_F_VN_GaussianFilterExp [ST]: FB_init, Clone, OnExecute, PreExecutionCheck
      function block Node_F_VN_LaplacianFilter [ST]: FB_init, Clone, OnExecute, PreExecutionCheck
      function block Node_F_VN_LaplacianFilterExp [ST]: FB_init, Clone, OnExecute, PreExecutionCheck
      function block Node_F_VN_LocalMaxima [ST]: FB_init, Clone, OnExecute, PreExecutionCheck
      function block Node_F_VN_LocalMinima [ST]: FB_init, Clone, OnExecute, PreExecutionCheck
      function block Node_F_VN_MedianFilter [ST]: FB_init, Clone, OnExecute, PreExecutionCheck
      function block Node_F_VN_MorphologicalOperator [ST]: FB_init, Clone, OnExecute, PreExecutionCheck
      function block Node_F_VN_RemoveLocalMaxima [ST]: FB_init, Clone, OnExecute, PreExecutionCheck
      function block Node_F_VN_RemoveLocalMinima [ST]: FB_init, Clone, OnExecute, PreExecutionCheck
      function block Node_F_VN_ScharrFilter [ST]: FB_init, Clone, OnExecute, PreExecutionCheck
      function block Node_F_VN_ScharrFilterExp [ST]: FB_init, Clone, OnExecute, PreExecutionCheck
      function block Node_F_VN_SobelFilter [ST]: FB_init, Clone, OnExecute, PreExecutionCheck
      function block Node_F_VN_SobelFilterExp [ST]: FB_init, Clone, OnExecute, PreExecutionCheck
      function block Node_F_VN_VarianceFilter [ST]: FB_init, Clone, OnExecute, PreExecutionCheck
      function block Node_F_VN_VarianceFilterExp [ST]: FB_init, Clone, OnExecute, PreExecutionCheck
    Image Segmentation/
      function block Node_F_VN_AdaptiveThreshold [ST]: FB_init, Clone, OnExecute, PreExecutionCheck
      function block Node_F_VN_AdaptiveThresholdExp [ST]: FB_init, Clone, OnExecute, PreExecutionCheck
      function block Node_F_VN_CheckColorRange [ST]: FB_init, Clone, OnExecute, PreExecutionCheck
      function block Node_F_VN_DoubleThreshold [ST]: FB_init, Clone, OnExecute, PreExecutionCheck
      function block Node_F_VN_SauvolaThreshold [ST]: FB_init, Clone, OnExecute, PreExecutionCheck
      function block Node_F_VN_Threshold [ST]: FB_init, Clone, OnExecute, PreExecutionCheck
      function block Node_F_VN_WatershedSegmentationExp [ST]: FB_init, Clone, OnExecute, PreExecutionCheck
    Keypoint Features/
      function block Node_F_VN_FilterGoodMatches [ST]: FB_init, Clone, OnExecute, PreExecutionCheck
      function block Node_F_VN_FindReferenceKeyPointsInImage [ST]: FB_init, Clone, OnExecute, PreExecutionCheck
      function block Node_F_VN_FindReferenceKeyPointsInImageAKAZE [ST]: FB_init, Clone, OnExecute, PreExecutionCheck
      function block Node_F_VN_FindReferenceKeyPointsInImageAKAZEExp [ST]: FB_init, Clone, OnExecute, PreExecutionCheck
      function block Node_F_VN_FindReferenceKeyPointsInImageBRISK [ST]: FB_init, Clone, OnExecute, PreExecutionCheck
      function block Node_F_VN_FindReferenceKeyPointsInImageBRISKExp [ST]: FB_init, Clone, OnExecute, PreExecutionCheck
      function block Node_F_VN_FindReferenceKeyPointsInImageExp [ST]: FB_init, Clone, OnExecute, PreExecutionCheck
      function block Node_F_VN_FindReferenceKeyPointsInImageORB [ST]: FB_init, Clone, OnExecute, PreExecutionCheck
      function block Node_F_VN_FindReferenceKeyPointsInImageORBExp [ST]: FB_init, Clone, OnExecute, PreExecutionCheck
      function block Node_F_VN_GetMatchCoordinates [ST]: FB_init, Clone, OnExecute, PreExecutionCheck
      function block Node_F_VN_KeyPointsAGAST [ST]: FB_init, Clone, OnExecute, PreExecutionCheck
      function block Node_F_VN_KeyPointsAGASTExp [ST]: FB_init, Clone, OnExecute, PreExecutionCheck
      function block Node_F_VN_KeyPointsAndDescriptorsAKAZE [ST]: FB_init, Clone, OnExecute, PreExecutionCheck
      function block Node_F_VN_KeyPointsAndDescriptorsAKAZEExp [ST]: FB_init, Clone, OnExecute, PreExecutionCheck
      function block Node_F_VN_KeyPointsAndDescriptorsBRISK [ST]: FB_init, Clone, OnExecute, PreExecutionCheck
      function block Node_F_VN_KeyPointsAndDescriptorsBRISKExp [ST]: FB_init, Clone, OnExecute, PreExecutionCheck
      function block Node_F_VN_KeyPointsAndDescriptorsKAZE [ST]: FB_init, Clone, OnExecute, PreExecutionCheck
      function block Node_F_VN_KeyPointsAndDescriptorsKAZEExp [ST]: FB_init, Clone, OnExecute, PreExecutionCheck
      function block Node_F_VN_KeyPointsAndDescriptorsORB [ST]: FB_init, Clone, OnExecute, PreExecutionCheck
      function block Node_F_VN_KeyPointsAndDescriptorsORBExp [ST]: FB_init, Clone, OnExecute, PreExecutionCheck
      function block Node_F_VN_KeyPointsFAST [ST]: FB_init, Clone, OnExecute, PreExecutionCheck
      function block Node_F_VN_KeyPointsFASTExp [ST]: FB_init, Clone, OnExecute, PreExecutionCheck
      function block Node_F_VN_KeyPointsGFTT [ST]: FB_init, Clone, OnExecute, PreExecutionCheck
      function block Node_F_VN_KeyPointsGFTTExp [ST]: FB_init, Clone, OnExecute, PreExecutionCheck
      function block Node_F_VN_KeyPointsMSER [ST]: FB_init, Clone, OnExecute, PreExecutionCheck
      function block Node_F_VN_KeyPointsMSERExp [ST]: FB_init, Clone, OnExecute, PreExecutionCheck
      function block Node_F_VN_KeyPointsSB [ST]: FB_init, Clone, OnExecute, PreExecutionCheck
      function block Node_F_VN_KeyPointsSBExp [ST]: FB_init, Clone, OnExecute, PreExecutionCheck
      function block Node_F_VN_MatchDescriptorsBF [ST]: FB_init, Clone, OnExecute, PreExecutionCheck
      function block Node_F_VN_MatchDescriptorsBFExp [ST]: FB_init, Clone, OnExecute, PreExecutionCheck
      function block Node_F_VN_MatchDescriptorsFlannLsh [ST]: FB_init, Clone, OnExecute, PreExecutionCheck
      function block Node_F_VN_MatchDescriptorsFlannLshExp [ST]: FB_init, Clone, OnExecute, PreExecutionCheck
      function block Node_F_VN_MatchDescriptorsKnnBF [ST]: FB_init, Clone, OnExecute, PreExecutionCheck
      function block Node_F_VN_MatchDescriptorsKnnBFExp [ST]: FB_init, Clone, OnExecute, PreExecutionCheck
      function block Node_F_VN_MatchDescriptorsKnnFlannLsh [ST]: FB_init, Clone, OnExecute, PreExecutionCheck
      function block Node_F_VN_MatchDescriptorsKnnFlannLshExp [ST]: FB_init, Clone, OnExecute, PreExecutionCheck
      function block Node_F_VN_RegionsMSER [ST]: FB_init, Clone, OnExecute, PreExecutionCheck
      function block Node_F_VN_RegionsMSERExp [ST]: FB_init, Clone, OnExecute, PreExecutionCheck
    Machine Learning/
    Measurement/
      function block Node_F_VN_AdjustSearchWindowOrientationToLinearEdge [ST]: FB_init, Clone, OnExecute, PreExecutionCheck
      function block Node_F_VN_ClosestPointsBF [ST]: FB_init, Clone, OnExecute, PreExecutionCheck
      function block Node_F_VN_LocateAxisAlignedEdges [ST]: FB_init, Clone, OnExecute, PreExecutionCheck
      function block Node_F_VN_LocateAxisAlignedEdgesExp [ST]: FB_init, Clone, OnExecute, PreExecutionCheck
      function block Node_F_VN_LocateCircularArc [ST]: FB_init, Clone, OnExecute, PreExecutionCheck
      function block Node_F_VN_LocateCircularArcExp [ST]: FB_init, Clone, OnExecute, PreExecutionCheck
      function block Node_F_VN_LocateCircularArcExp2 [ST]: FB_init, Clone, OnExecute, PreExecutionCheck
      function block Node_F_VN_LocateEdge [ST]: FB_init, Clone, OnExecute, PreExecutionCheck
      function block Node_F_VN_LocateEdgeExp [ST]: FB_init, Clone, OnExecute, PreExecutionCheck
      function block Node_F_VN_LocateEdgeExp2 [ST]: FB_init, Clone, OnExecute, PreExecutionCheck
      function block Node_F_VN_LocateEdges [ST]: FB_init, Clone, OnExecute, PreExecutionCheck
      function block Node_F_VN_LocateEdgesExp [ST]: FB_init, Clone, OnExecute, PreExecutionCheck
      function block Node_F_VN_LocateEdgesExp2 [ST]: FB_init, Clone, OnExecute, PreExecutionCheck
      function block Node_F_VN_LocateEllipse [ST]: FB_init, Clone, OnExecute, PreExecutionCheck
      function block Node_F_VN_LocateEllipseExp [ST]: FB_init, Clone, OnExecute, PreExecutionCheck
      function block Node_F_VN_LocateEllipseExp2 [ST]: FB_init, Clone, OnExecute, PreExecutionCheck
      function block Node_F_VN_MeasureAngleBetweenEdges [ST]: FB_init, Clone, OnExecute, PreExecutionCheck
      function block Node_F_VN_MeasureAngleBetweenEdgesExp [ST]: FB_init, Clone, OnExecute, PreExecutionCheck
      function block Node_F_VN_MeasureAngleBetweenEdgesExp2 [ST]: FB_init, Clone, OnExecute, PreExecutionCheck
      function block Node_F_VN_MeasureEdgeDistance [ST]: FB_init, Clone, OnExecute, PreExecutionCheck
      function block Node_F_VN_MeasureEdgeDistanceExp [ST]: FB_init, Clone, OnExecute, PreExecutionCheck
      function block Node_F_VN_MeasureEdgeDistanceExp2 [ST]: FB_init, Clone, OnExecute, PreExecutionCheck
      function block Node_F_VN_MeasureMinEdgeDistance [ST]: FB_init, Clone, OnExecute, PreExecutionCheck
      function block Node_F_VN_MeasureMinEdgeDistanceExp [ST]: FB_init, Clone, OnExecute, PreExecutionCheck
      function block Node_F_VN_MeasureMinEdgeDistanceExp2 [ST]: FB_init, Clone, OnExecute, PreExecutionCheck
    Miscellaneous/
      function block Node_F_VN_CheckFunctionInitialization [ST]: FB_init, Clone, OnExecute, PreExecutionCheck
      function block Node_F_VN_ClipLineToBoundary [ST]: FB_init, Clone, OnExecute, PreExecutionCheck
      function block Node_F_VN_ClipLineToBoundary_ITcVnImage [ST]: FB_init, Clone, OnExecute, PreExecutionCheck
      function block Node_F_VN_ClipLineToBoundary_TcVnRectangle_DINT [ST]: FB_init, Clone, OnExecute, PreExecutionCheck
      function block Node_F_VN_DeinitializeFunction [ST]: FB_init, Clone, OnExecute, PreExecutionCheck
      function block Node_F_VN_HuMomentInvariants [ST]: FB_init, Clone, OnExecute, PreExecutionCheck
      function block Node_F_VN_InvertMatrix3x3 [ST]: FB_init, Clone, OnExecute, PreExecutionCheck
      function block Node_F_VN_LineIntersectionPoint [ST]: FB_init, Clone, OnExecute, PreExecutionCheck
      function block Node_F_VN_LineIntersectionPointAndAngle [ST]: FB_init, Clone, OnExecute, PreExecutionCheck
      function block Node_F_VN_OrthogonalVector_TcVnVector2_DINT [ST]: FB_init, Clone, OnExecute, PreExecutionCheck
      function block Node_F_VN_OrthogonalVector_TcVnVector2_LREAL [ST]: FB_init, Clone, OnExecute, PreExecutionCheck
      function block Node_F_VN_OrthogonalVector_TcVnVector2_REAL [ST]: FB_init, Clone, OnExecute, PreExecutionCheck
      function block Node_F_VN_PointToLineDistance_TcVnPoint2_DINT [ST]: FB_init, Clone, OnExecute, PreExecutionCheck
      function block Node_F_VN_PointToLineDistance_TcVnPoint2_LREAL [ST]: FB_init, Clone, OnExecute, PreExecutionCheck
      function block Node_F_VN_PointToLineDistance_TcVnPoint2_REAL [ST]: FB_init, Clone, OnExecute, PreExecutionCheck
      function block Node_F_VN_PointToPointDirection_TcVnPoint2_DINT [ST]: FB_init, Clone, OnExecute, PreExecutionCheck
      function block Node_F_VN_PointToPointDirection_TcVnPoint2_LREAL [ST]: FB_init, Clone, OnExecute, PreExecutionCheck
      function block Node_F_VN_PointToPointDirection_TcVnPoint2_REAL [ST]: FB_init, Clone, OnExecute, PreExecutionCheck
      function block Node_F_VN_PointToPointDistance_TcVnPoint2_DINT [ST]: FB_init, Clone, OnExecute, PreExecutionCheck
      function block Node_F_VN_PointToPointDistance_TcVnPoint2_LREAL [ST]: FB_init, Clone, OnExecute, PreExecutionCheck
      function block Node_F_VN_PointToPointDistance_TcVnPoint2_REAL [ST]: FB_init, Clone, OnExecute, PreExecutionCheck
      function block Node_F_VN_RotatedRectangleCorners [ST]: FB_init, Clone, OnExecute, PreExecutionCheck
      function block Node_F_VN_RotatedRectangleIntersection [ST]: FB_init, Clone, OnExecute, PreExecutionCheck
    Neural Network/
      function block Node_F_VN_Reduce [ST]: FB_init, Clone, OnExecute, PreExecutionCheck
      function block Node_F_VN_ReduceArg [ST]: FB_init, Clone, OnExecute, PreExecutionCheck
      function block Node_F_VN_Sigmoid [ST]: FB_init, Clone, OnExecute, PreExecutionCheck
      function block Node_F_VN_SigmoidExp [ST]: FB_init, Clone, OnExecute, PreExecutionCheck
      function block Node_F_VN_SoftMax [ST]: FB_init, Clone, OnExecute, PreExecutionCheck
    OCR/
      function block Node_F_VN_OCR [ST]: FB_init, Clone, OnExecute, PreExecutionCheck
      function block Node_F_VN_OCRExp [ST]: FB_init, Clone, OnExecute, PreExecutionCheck
    Polarization/
      function block Node_F_VN_AngleAndDegreeOfLinearPolarization [ST]: FB_init, Clone, OnExecute, PreExecutionCheck
      function block Node_F_VN_DemosaicPolarizedImage [ST]: FB_init, Clone, OnExecute, PreExecutionCheck
      function block Node_F_VN_PolarizedImageGlareReduction [ST]: FB_init, Clone, OnExecute, PreExecutionCheck
    Texture Analysis/
      function block Node_F_VN_Granulometry [ST]: FB_init, Clone, OnExecute, PreExecutionCheck
      function block Node_F_VN_HaralickFeatures [ST]: FB_init, Clone, OnExecute, PreExecutionCheck
    VisionNode/
      function block VisionHardwareNode [ST]: Execute, PreExecutionCheck
      function block VisionNode [ST]: Execute, PreExecutionCheck
    function block VisionNodePack [ST]: RegisterWithNodeFactory
  global variables GVL_COLOURS
  function block VisionPack [ST]: Register
*)

// GVL_COLOURS
{attribute 'qualified_only'}
VAR_GLOBAL
    RGBA_BLACK    : TcVnVector4_LREAL := [0, 0, 0, 255];
    RGBA_RED      : TcVnVector4_LREAL := [255, 0, 0, 255];
    RGBA_YELLOW   : TcVnVector4_LREAL := [255, 255, 0, 255];
    RGBA_GREEN    : TcVnVector4_LREAL := [0, 255, 0, 255];
    RGBA_CYAN     : TcVnVector4_LREAL := [0, 255, 255, 255];
    RGBA_BLUE     : TcVnVector4_LREAL := [0, 0, 255, 255];
    RGBA_MAGENTA  : TcVnVector4_LREAL := [255, 0, 255, 255];
    RGBA_WHITE    : TcVnVector4_LREAL := [255, 255, 255, 255];
    RGBA_RANDOM   : TcVnVector4_LREAL := [-1, -1, -1, -1];
END_VAR

// Datatypes/Aliases/_GVCP_REGISTER_ADDRESS
{attribute 'linkalways'} 
{attribute 'no_explicit_call' := 'This FB is a CLASS and must be accessed using methods or properties'}
{attribute 'enable_dynamic_creation'}
FUNCTION_BLOCK _GVCP_REGISTER_ADDRESS EXTENDS AliasDatatypeBase
VAR
	localData : GVCP_REGISTER_ADDRESS;
	activeData : REFERENCE TO GVCP_REGISTER_ADDRESS REF= localData;
	aliasBaseDatatype : _UDINT(0);
END_VAR

METHOD PROTECTED SetBaseDatatypeReference
VAR_INPUT
END_VAR
aliasBaseDatatype.MakeReferenceTo(activeData);
END_METHOD

PROPERTY PUBLIC Address : PVOID
GET
Address := ADR(activeData);
END_GET
END_PROPERTY

METHOD PUBLIC ClearReference
VAR_INPUT
END_VAR
activeData REF= localData;
SetBaseDatatypeReference();
END_METHOD

PROPERTY PUBLIC Size : UDINT
GET
Size := SIZEOF(activeData);
END_GET
END_PROPERTY

METHOD FB_init : BOOL
VAR_INPUT
	bInitRetains : BOOL; // if TRUE, the retain variables are initialized (warm start / cold start)
	bInCopyCode : BOOL;  // if TRUE, the instance afterwards gets moved into the copy code (online change)
	InitialValue : GVCP_REGISTER_ADDRESS; // if possible, not all values can be initialized
END_VAR
localData := InitialValue;
SetBaseDatatypeReference();
AddBaseDatatype(aliasBaseDatatype);
END_METHOD

METHOD PUBLIC Clone : I_Datatype
VAR
    pClone : POINTER TO _GVCP_REGISTER_ADDRESS;
END_VAR
pClone := __NEW(_GVCP_REGISTER_ADDRESS(InitialValue := Value));
Clone := pClone^;
END_METHOD

PROPERTY PUBLIC Identifier : T_MAXSTRING
GET
Identifier := 'GVCP_REGISTER_ADDRESS';
END_GET
END_PROPERTY

METHOD PUBLIC MakeReferenceTo
VAR_INPUT
	ReferenceTarget : REFERENCE TO GVCP_REGISTER_ADDRESS;
END_VAR
activeData REF= ReferenceTarget;
SetBaseDatatypeReference();
END_METHOD

METHOD TryMakeReferenceTo : BOOL
VAR_INPUT
	Target : I_Datatype;
END_VAR
VAR
	pTargetData : POINTER TO GVCP_REGISTER_ADDRESS;
END_VAR
IF NOT IsEquivalentTo(Target) THEN
	RETURN;
END_IF

pTargetData := Target.Address;
activeData REF= pTargetData^;
SetBaseDatatypeReference();
TryMakeReferenceTo := TRUE;
END_METHOD

PROPERTY PUBLIC Value : REFERENCE TO GVCP_REGISTER_ADDRESS
GET
Value REF= activeData;
END_GET
END_PROPERTY

END_FUNCTION_BLOCK

// Datatypes/Aliases/_GVCP_REGISTER_VALUE
{attribute 'linkalways'}
{attribute 'no_explicit_call' := 'This FB is a CLASS and must be accessed using methods or properties'}
{attribute 'enable_dynamic_creation'}
FUNCTION_BLOCK _GVCP_REGISTER_VALUE EXTENDS AliasDatatypeBase
VAR
	localData : GVCP_REGISTER_VALUE;
	activeData : REFERENCE TO GVCP_REGISTER_VALUE REF= localData;
	aliasBaseDatatype : _UDINT(0);
END_VAR

METHOD PROTECTED SetBaseDatatypeReference
VAR_INPUT
END_VAR
aliasBaseDatatype.MakeReferenceTo(activeData);
END_METHOD

PROPERTY PUBLIC Address : PVOID
GET
Address := ADR(activeData);
END_GET
END_PROPERTY

METHOD PUBLIC ClearReference
VAR_INPUT
END_VAR
activeData REF= localData;
SetBaseDatatypeReference();
END_METHOD

PROPERTY PUBLIC Size : UDINT
GET
Size := SIZEOF(activeData);
END_GET
END_PROPERTY

METHOD FB_init : BOOL
VAR_INPUT
	bInitRetains : BOOL; // if TRUE, the retain variables are initialized (warm start / cold start)
	bInCopyCode : BOOL;  // if TRUE, the instance afterwards gets moved into the copy code (online change)
	InitialValue : GVCP_REGISTER_VALUE := 0;
END_VAR
localData := InitialValue;
SetBaseDatatypeReference();
AddBaseDatatype(aliasBaseDatatype);
END_METHOD

METHOD PUBLIC Clone : I_Datatype
VAR
    pClone : POINTER TO _GVCP_REGISTER_VALUE;
END_VAR
pClone := __NEW(_GVCP_REGISTER_VALUE(InitialValue := Value));
IF pClone = 0 THEN
    RETURN;
END_IF
pClone^.TryCopyFrom(THIS^);
Clone := pClone^;
END_METHOD

PROPERTY PUBLIC Identifier : T_MAXSTRING
GET
Identifier := 'GVCP_REGISTER_VALUE';
END_GET
END_PROPERTY

METHOD PUBLIC MakeReferenceTo
VAR_INPUT
	ReferenceTarget : REFERENCE TO GVCP_REGISTER_VALUE;
END_VAR
activeData REF= ReferenceTarget;
SetBaseDatatypeReference();
END_METHOD

METHOD TryMakeReferenceTo : BOOL
VAR_INPUT
	Target : I_Datatype;
END_VAR
VAR
	pTargetData : POINTER TO GVCP_REGISTER_VALUE;
END_VAR
IF NOT IsEquivalentTo(Target) THEN
	RETURN;
END_IF

pTargetData := Target.Address;
activeData REF= pTargetData^;
SetBaseDatatypeReference();
TryMakeReferenceTo := TRUE;
END_METHOD

PROPERTY PUBLIC Value : REFERENCE TO GVCP_REGISTER_VALUE
GET
Value REF= activeData;
END_GET
END_PROPERTY

END_FUNCTION_BLOCK

// Datatypes/Aliases/_TcVnArray10_ITcVnImage
{attribute 'linkalways'} 
{attribute 'no_explicit_call' := 'This FB is a CLASS and must be accessed using methods or properties'}
{attribute 'enable_dynamic_creation'}
FUNCTION_BLOCK _TcVnArray10_ITcVnImage EXTENDS AliasDatatypeBase
VAR
	localData : TcVnArray10_ITcVnImage;
	activeData : REFERENCE TO TcVnArray10_ITcVnImage REF= localData;
	aliasBaseDatatype : _Array0to9OfITcVnImage;
END_VAR

METHOD PROTECTED SetBaseDatatypeReference
VAR_INPUT
END_VAR
aliasBaseDatatype.MakeReferenceTo(activeData);
END_METHOD

PROPERTY PUBLIC Address : PVOID
GET
Address := ADR(activeData);
END_GET
END_PROPERTY

METHOD PUBLIC ClearReference
VAR_INPUT
END_VAR
activeData REF= localData;
SetBaseDatatypeReference();
END_METHOD

PROPERTY PUBLIC Size : UDINT
GET
Size := SIZEOF(activeData);
END_GET
END_PROPERTY

METHOD FB_init : BOOL
VAR_INPUT
	bInitRetains : BOOL; // if TRUE, the retain variables are initialized (warm start / cold start)
	bInCopyCode : BOOL;  // if TRUE, the instance afterwards gets moved into the copy code (online change)
	//InitialValue : TcVnArray10_ITcVnImage; // if possible, not all values can be initialized
END_VAR
//localData := InitialValue; // if possible, not all values can be initialized
SetBaseDatatypeReference();
AddBaseDatatype(aliasBaseDatatype);
END_METHOD

METHOD PUBLIC Clone : I_Datatype
VAR
    pClone : POINTER TO _TcVnArray10_ITcVnImage;
END_VAR
pClone := __NEW(_TcVnArray10_ITcVnImage);
Clone := pClone^;
END_METHOD

PROPERTY PUBLIC Identifier : T_MAXSTRING
GET
Identifier := 'TcVnArray10_ITcVnImage';
END_GET
END_PROPERTY

METHOD PUBLIC MakeReferenceTo
VAR_INPUT
	ReferenceTarget : REFERENCE TO TcVnArray10_ITcVnImage;
END_VAR
activeData REF= ReferenceTarget;
SetBaseDatatypeReference();
END_METHOD

METHOD TryMakeReferenceTo : BOOL
VAR_INPUT
	Target : I_Datatype;
END_VAR
VAR
	pTargetData : POINTER TO TcVnArray10_ITcVnImage;
END_VAR
IF NOT IsEquivalentTo(Target) THEN
	RETURN;
END_IF

pTargetData := Target.Address;
activeData REF= pTargetData^;
SetBaseDatatypeReference();
TryMakeReferenceTo := TRUE;
END_METHOD

PROPERTY PUBLIC Value : REFERENCE TO TcVnArray10_ITcVnImage
GET
Value REF= activeData;
END_GET
END_PROPERTY

END_FUNCTION_BLOCK

// Datatypes/Arrays/_Array0to9OfITcVnImage
{attribute 'linkalways'} 
{attribute 'no_explicit_call' := 'This FB is a CLASS and must be accessed using methods or properties'}
{attribute 'enable_dynamic_creation'}
FUNCTION_BLOCK _Array0to9OfITcVnImage EXTENDS ArrayDatatypeBase_1D
VAR CONSTANT
	lBound : DINT := 0;
	uBound : DINT := 9;
END_VAR
VAR
	localData : ARRAY [lBound..uBound] OF ITcVnImage;
	activeData : REFERENCE TO ARRAY [lBound..uBound] OF ITcVnImage REF= localData;
	elements : ARRAY [lBound..uBound] OF _ITcVnImage;
	baseType : _ITcVnImage;
END_VAR

METHOD FB_init : BOOL
VAR_INPUT
	bInitRetains : BOOL; // if TRUE, the retain variables are initialized (warm start / cold start)
	bInCopyCode : BOOL;  // if TRUE, the instance afterwards gets moved into the copy code (online change)
END_VAR
SetElementReference();
END_METHOD

METHOD PROTECTED OnSerializeArrayValues
VAR_INPUT
	Serializer : I_Serializer;
END_VAR
VAR
	i : DINT;
END_VAR
FOR i := lBound TO uBound DO
	elements[i].SerializeWith(Serializer);
END_FOR
END_METHOD

METHOD PROTECTED SetElementReference
VAR_INPUT
END_VAR
VAR
	i : DINT;
END_VAR
FOR i := lBound TO uBound DO
	elements[i].MakeReferenceTo(activeData[i]);
END_FOR
END_METHOD

METHOD PROTECTED TryDeserializeArrayValues : BOOL
VAR_INPUT
	Deserializer : I_Deserializer;
	Feedback : I_DeserializerFeedback;
END_VAR
VAR
	enumerator : I_DeserializerArrayForwardEnumerator;
	i : DINT;
END_VAR
enumerator := Deserializer.GetArrayEnumerator();
i := lBound;

WHILE enumerator.MoveNext() AND i <= uBound DO
	
	IF NOT elements[i].TryDeserializeFrom(enumerator.Current, Feedback) THEN
		EXIT;
	END_IF
	i := i + 1;

END_WHILE
enumerator.Dispose();
END_METHOD

PROPERTY PUBLIC Address : PVOID
GET
Address := ADR(activeData);
END_GET
END_PROPERTY

PROPERTY PUBLIC BaseDatatype : I_Datatype
GET
BaseDatatype := baseType;
END_GET
END_PROPERTY

METHOD PUBLIC ClearReference
VAR_INPUT
END_VAR
activeData REF= localData;
SetElementReference();
END_METHOD

PROPERTY PUBLIC Size : UDINT
GET
Size := SIZEOF(activeData);
END_GET
END_PROPERTY

METHOD PUBLIC TryGetElementAsDatatypeByIndex : BOOL
VAR_INPUT
	Index : DINT;
	Destination : REFERENCE TO I_Datatype;
END_VAR
IF Index < lbound OR Index > ubound THEN
	RETURN;
END_IF

Destination := elements[Index];
TryGetElementAsDatatypeByIndex := TRUE;
END_METHOD

METHOD PUBLIC TryGetLowerBound : BOOL
VAR_INPUT
	Dimention : UDINT;
	Destination : REFERENCE TO DINT;
END_VAR
IF Dimention = 1 THEN
	Destination := lBound;
	TryGetLowerBound := TRUE;
END_IF
END_METHOD

METHOD PUBLIC TryGetUpperBound : BOOL
VAR_INPUT
	Dimention : UDINT;
	Destination : REFERENCE TO DINT;
END_VAR
IF Dimention = 1 THEN
	Destination := uBound;
	TryGetUpperBound := TRUE;
END_IF
END_METHOD

METHOD PUBLIC Clone : I_Datatype
VAR
    pClone : POINTER TO _Array0to9OfITcVnImage;
END_VAR
pClone := __NEW(_Array0to9OfITcVnImage());
pClone^.Value := Value;
Clone := pClone^;
END_METHOD

METHOD PUBLIC MakeReferenceTo
VAR_INPUT
	ReferenceTarget : REFERENCE TO ARRAY [lBound..uBound] OF ITcVnImage;
END_VAR
activeData REF= ReferenceTarget;
SetElementReference();
END_METHOD

METHOD TryMakeReferenceTo : BOOL
VAR_INPUT
	Target : I_Datatype;
END_VAR
VAR
	pTargetData : POINTER TO ARRAY [lBound..uBound] OF ITcVnImage;
END_VAR
IF NOT IsEquivalentTo(Target) THEN
	RETURN;
END_IF

pTargetData := Target.Address;
activeData REF= pTargetData^;
SetElementReference();
TryMakeReferenceTo := TRUE;
END_METHOD

PROPERTY PUBLIC Value : REFERENCE TO ARRAY [lBound..uBound] OF ITcVnImage;
GET
Value ref= activeData;
END_GET
END_PROPERTY

END_FUNCTION_BLOCK

// Datatypes/Interfaces/Images/ITcVnImage/_ITcVnImage
{attribute 'linkalways'} 
{attribute 'no_explicit_call' := 'This FB is a CLASS and must be accessed using methods or properties'}
{attribute 'enable_dynamic_creation'}
FUNCTION_BLOCK _ITcVnImage EXTENDS InterfaceDatatypeBase IMPLEMENTS I_InterfaceDatatype_ITcVnImage
VAR
	localData : ITcVnImage;
	activeData : REFERENCE TO ITcVnImage REF= localData;
END_VAR

PROPERTY PUBLIC Address : PVOID
GET
Address := ADR(activeData);
END_GET
END_PROPERTY

METHOD PUBLIC ClearReference
VAR_INPUT
END_VAR
activeData REF= localData;
END_METHOD

PROPERTY PUBLIC Size : UDINT
GET
Size := SIZEOF(activeData);
END_GET
END_PROPERTY

METHOD FB_exit : BOOL
VAR_INPUT
	bInCopyCode : BOOL; // if TRUE, the exit method is called for exiting an instance that is copied afterwards (online change).
END_VAR
IF bInCopyCode THEN
	RETURN;
END_IF

TryTcReleaseLocal();
END_METHOD

METHOD PRIVATE TryGetElementTypeFromInfo : BOOL;
VAR_INPUT
	ImageInfo : TcVnImageInfo;
	Destination : REFERENCE TO ETcVnElementType;
END_VAR
CASE ImageInfo.stPixelFormat.nElementSize OF
	
	8 : // 8bit
	
		IF ImageInfo.stPixelFormat.bSigned THEN
			Destination := ETcVnElementType.TCVN_ET_SINT;
		ELSE	
			Destination := ETcVnElementType.TCVN_ET_USINT;
		END_IF
		TryGetElementTypeFromInfo := TRUE;
	
	16 : // 16bit
	
		IF ImageInfo.stPixelFormat.bSigned THEN
			Destination := ETcVnElementType.TCVN_ET_INT;
		ELSE	
			Destination := ETcVnElementType.TCVN_ET_UINT;
		END_IF
		TryGetElementTypeFromInfo := TRUE;
	
	32 : // 32bit
	
		IF ImageInfo.stPixelFormat.bSigned AND NOT ImageInfo.stPixelFormat.bFloat THEN
			Destination := ETcVnElementType.TCVN_ET_DINT;
			TryGetElementTypeFromInfo := TRUE;
		END_IF
		
		IF ImageInfo.stPixelFormat.bFloat THEN
			Destination := ETcVnElementType.TCVN_ET_REAL;
			TryGetElementTypeFromInfo := TRUE;
		END_IF
		
	64 : // 64bit
	
		IF ImageInfo.stPixelFormat.bFloat THEN
			Destination := ETcVnElementType.TCVN_ET_LREAL;
			TryGetElementTypeFromInfo := TRUE;
		END_IF
		
ELSE
	
	RETURN;

END_CASE
END_METHOD

METHOD PUBLIC TryTcReleaseLocal : BOOL
VAR_INPUT
END_VAR
IF localData = 0 THEN
	RETURN;
END_IF

IF localData.TcRelease() = 0 THEN
	localData := 0;
END_IF

TryTcReleaseLocal := TRUE;
END_METHOD

METHOD PUBLIC Clone : I_Datatype
VAR
    pClone : POINTER TO _ITcVnImage;
END_VAR
pClone := __NEW(_ITcVnImage);
Clone := pClone^;
END_METHOD

PROPERTY PUBLIC Identifier : T_MAXSTRING
GET
Identifier := 'ITcVnImage';
END_GET
END_PROPERTY

METHOD PUBLIC MakeReferenceTo
VAR_INPUT
	ReferenceTarget : REFERENCE TO ITcVnImage;
END_VAR
activeData REF= ReferenceTarget;
END_METHOD

METHOD PUBLIC SerializeWith
VAR_INPUT
	Serializer : I_Serializer;
END_VAR
VAR
	result: HRESULT;
	exportImageSize: ULINT;
	buffer : POINTER TO BYTE;
	imageInfo : _TcVnImageInfo;
END_VAR
IF NOT (activeData <> 0) THEN
	// no image available, so drop out.. need to add serialization?
	Serializer.AddNull();
	RETURN;
END_IF

result := F_VN_ExportImageSize(ipImage:=activeData, nBufferSize:=exportImageSize, hrPrev:=result);

IF FAILED(result) THEN
	// export to bmp size failed, so drop out.. need to add serialization?
	Serializer.AddNull();
	RETURN;
END_IF

IF exportImageSize > DatatypeLimits.UDINT_MAX_VALUE THEN
	// export is too big for __NEW, so drop out..
	Serializer.AddNull();
	RETURN;
END_IF

IF exportImageSize <= 0 THEN
	// export is zero size, so drop out.. 
	Serializer.AddNull();
	RETURN;
END_IF
	
buffer := __NEW(BYTE,ULINT_TO_UDINT(exportImageSize));
result := F_VN_ExportImage(ipImage:=activeData, pBuffer:=buffer, nBufferSize:=exportImageSize, hrPrev:=result);

IF FAILED(result) THEN
	// export to bmp failed, so drop out.. 
	Serializer.AddNull();
	__DELETE(buffer);
	RETURN;
END_IF

activeData.GetImageInfo(imageInfo.value);

Serializer.StartObject();
Serializer.AddKeyObject('imageInfo',imageInfo);
Serializer.AddKey('imageData');
Serializer.AddBase64(buffer,ULINT_TO_DINT(exportImageSize));
Serializer.EndObject();

__DELETE(buffer);
END_METHOD

METHOD TryMakeReferenceTo : BOOL
VAR_INPUT
	Target : I_Datatype;
END_VAR
VAR
	pTargetData : POINTER TO ITcVnImage;
END_VAR
IF NOT IsEquivalentTo(Target) THEN
	RETURN;
END_IF

pTargetData := Target.Address;
activeData REF= pTargetData^;
TryMakeReferenceTo := TRUE;
END_METHOD

PROPERTY PUBLIC Value : REFERENCE TO ITcVnImage
GET
Value REF= activeData;
END_GET
END_PROPERTY

METHOD PUBLIC HasChannelCount : BOOL
VAR_INPUT
	ChannelCount : BYTE;
END_VAR
VAR
    pixelFormat : TcVnPixelFormat;
END_VAR
IF NOT TryGetPixelFormat(pixelFormat) THEN
    RETURN;
END_IF

IF NOT (pixelFormat.nChannels = ChannelCount) THEN
    RETURN;
END_IF

HasChannelCount := TRUE;
END_METHOD

METHOD PUBLIC IsElementType : BOOL
VAR_INPUT
	ElementType : ETcVnElementType;
END_VAR
VAR
    pixelFormat : TcVnPixelFormat;
END_VAR
IF NOT TryGetPixelFormat(pixelFormat) THEN
    RETURN;
END_IF

CASE elementType OF

    TCVN_ET_USINT:
        IF pixelFormat.bFloat THEN
            RETURN;
        END_IF
        IF pixelFormat.bSigned THEN
            RETURN;
        END_IF
        IF NOT (pixelFormat.nElementSize = 8) THEN
            RETURN;
        END_IF
        IsElementType := TRUE;

    TCVN_ET_SINT:
        IF pixelFormat.bFloat THEN
            RETURN;
        END_IF
        IF NOT pixelFormat.bSigned THEN
            RETURN;
        END_IF
        IF NOT (pixelFormat.nElementSize = 8) THEN
            RETURN;
        END_IF
        IsElementType := TRUE;

    TCVN_ET_UINT:
        IF pixelFormat.bFloat THEN
            RETURN;
        END_IF
        IF pixelFormat.bSigned THEN
            RETURN;
        END_IF
        IF NOT (pixelFormat.nElementSize = 16) THEN
            RETURN;
        END_IF
        IsElementType := TRUE;

    TCVN_ET_INT:
        IF pixelFormat.bFloat THEN
            RETURN;
        END_IF
        IF NOT pixelFormat.bSigned THEN
            RETURN;
        END_IF
        IF NOT (pixelFormat.nElementSize = 16) THEN
            RETURN;
        END_IF
        IsElementType := TRUE;

    TCVN_ET_DINT:
        IF pixelFormat.bFloat THEN
            RETURN;
        END_IF
        IF NOT pixelFormat.bSigned THEN
            RETURN;
        END_IF
        IF NOT (pixelFormat.nElementSize = 32) THEN
            RETURN;
        END_IF
        IsElementType := TRUE;

    TCVN_ET_REAL:
        IF NOT pixelFormat.bFloat THEN
            RETURN;
        END_IF
        IF NOT (pixelFormat.nElementSize = 32) THEN
            RETURN;
        END_IF
        IsElementType := TRUE;

    TCVN_ET_LREAL:
        IF NOT pixelFormat.bFloat THEN
            RETURN;
        END_IF
        IF NOT (pixelFormat.nElementSize = 64) THEN
            RETURN;
        END_IF
        IsElementType := TRUE;

END_CASE
END_METHOD

METHOD PUBLIC IsPixelDepth : BOOL
VAR_INPUT
	PixelDepth : UINT;
END_VAR
VAR
    pixelFormat : TcVnPixelFormat;
END_VAR
IF NOT TryGetPixelFormat(pixelFormat) THEN
    RETURN;
END_IF

IF NOT (pixelFormat.nElementSize = PixelDepth) THEN
    RETURN;
END_IF

IsPixelDepth := TRUE;
END_METHOD

PROPERTY PUBLIC IsValid : BOOL
GET
IsValid := activeData <> 0;
END_GET
END_PROPERTY

METHOD PUBLIC TryCopyContentFrom : BOOL
VAR_INPUT
	Source : I_InterfaceDatatype;
END_VAR
VAR
	ipSrcImage : I_InterfaceDatatype_ITcVnImage;
	hresult : HRESULT;
END_VAR
IF NOT __QUERYINTERFACE(Source, ipSrcImage) THEN
	RETURN;
END_IF

hresult := F_VN_CopyImage(
    ipSrcImage := ipSrcImage.Value,
	ipDestImage := Value,
	hrPrev:= S_OK);
    

TryCopyContentFrom := SUCCEEDED(hresult);
END_METHOD

METHOD TryDeserializeFrom : BOOL
VAR_INPUT
	Deserializer : I_Deserializer;
	Feedback : I_DeserializerFeedback;
END_VAR
VAR
	imageInfo : _TcVnImageInfo;
	imageSizeInBytes : UDINT;
	buffer : POINTER TO BYTE;
	hr : HRESULT;
	elementType : ETcVnElementType;
END_VAR
IF NOT Deserializer.TryDeserializeKeyToObject('imageInfo', imageInfo, Feedback) THEN
	RETURN;
END_IF

imageSizeInBytes := ULINT_TO_UDINT(imageInfo.nImageSize.Value);

IF imageSizeInBytes = 0 THEN
	TryDeserializeFrom := TRUE;
	RETURN;
END_IF

buffer := __NEW(BYTE, imageSizeInBytes);

IF NOT Deserializer.TryGetKeyBase64('imageData', buffer, UDINT_TO_DINT(imageSizeInBytes), Feedback) THEN
	__DELETE(buffer);
	RETURN;
END_IF

TryGetElementTypeFromInfo(imageInfo.Value, elementType);

hr := F_VN_CreateImageFromArray(
	pData := buffer,
	ipImage := activeData,
	nWidth := imageInfo.nWidth.Value,
	nHeight :=  imageInfo.nHeight.Value,
	ePixelType := elementType,
	nChannelNum := imageInfo.stPixelFormat.nChannels.Value, 
	hrPrev := hr);

__DELETE(buffer);

TryDeserializeFrom := TRUE;
END_METHOD

METHOD PUBLIC TryGetHeight : BOOL
VAR_INPUT
	Destination : REFERENCE TO UDINT;
END_VAR
IF NOT IsValid THEN
	RETURN;
END_IF

TryGetHeight := SUCCEEDED(activeData.GetHeight(Destination));
END_METHOD

METHOD PUBLIC TryGetImageData : BOOL
VAR_INPUT
	Destination : POINTER TO ITcVnData;
END_VAR
IF NOT IsValid THEN
	RETURN;
END_IF

TryGetImageData := SUCCEEDED(activeData.GetImageData(Destination));
END_METHOD

METHOD PUBLIC TryGetImageInfo : BOOL
VAR_INPUT
	Destination : REFERENCE TO  TcVnImageInfo;
END_VAR
IF NOT IsValid THEN
	RETURN;
END_IF

TryGetImageInfo := SUCCEEDED(activeData.GetImageInfo(Destination));
END_METHOD

METHOD PUBLIC TryGetImageSize : BOOL
VAR_INPUT
	Destination : REFERENCE TO ULINT;
END_VAR
IF NOT IsValid THEN
	RETURN;
END_IF

TryGetImageSize := SUCCEEDED(activeData.GetImageSize(Destination));
END_METHOD

METHOD PUBLIC TryGetPixelFormat : BOOL
VAR_INPUT
	Destination : REFERENCE TO  TcVnPixelFormat;
END_VAR
IF NOT IsValid THEN
	RETURN;
END_IF

TryGetPixelFormat := SUCCEEDED(activeData.GetPixelFormat(Destination));
END_METHOD

METHOD PUBLIC TryGetRowPointer : BOOL
VAR_INPUT
	RowIndex : UDINT;
	Destination : POINTER TO PVOID;
END_VAR
IF NOT IsValid THEN
	RETURN;
END_IF

TryGetRowPointer := SUCCEEDED(activeData.GetRowPointer(RowIndex, Destination));
END_METHOD

METHOD PUBLIC TryGetWidth : BOOL
VAR_INPUT
	Destination : REFERENCE TO UDINT;
END_VAR
IF NOT IsValid THEN
	RETURN;
END_IF

TryGetWidth := SUCCEEDED(activeData.GetWidth(Destination));
END_METHOD

METHOD PUBLIC TryGetXPadding : BOOL
VAR_INPUT
	Destination : REFERENCE TO UINT;
END_VAR
IF NOT IsValid THEN
	RETURN;
END_IF

TryGetXPadding := SUCCEEDED(activeData.GetXPadding(Destination));
END_METHOD

METHOD PUBLIC TryGetYPadding : BOOL
VAR_INPUT
	Destination : REFERENCE TO UINT;
END_VAR
IF NOT IsValid THEN
	RETURN;
END_IF

TryGetYPadding := SUCCEEDED(activeData.GetYPadding(Destination));
END_METHOD

METHOD PUBLIC TryReleaseRowPointer : BOOL
VAR_INPUT
	ppRow : POINTER TO PVOID;
END_VAR
IF NOT IsValid THEN
	RETURN;
END_IF

TryReleaseRowPointer := SUCCEEDED(activeData.ReleaseRowPointer(ppRow));
END_METHOD

METHOD PUBLIC TryTcAddRef : BOOL
VAR_INPUT
END_VAR
IF activeData = 0 THEN
	RETURN;
END_IF

IF activeData.TcAddRef() = 0 THEN
	activeData := 0;
END_IF

TryTcAddRef := TRUE;
END_METHOD

METHOD PUBLIC TryTcRelease : BOOL
VAR_INPUT
END_VAR
IF activeData = 0 THEN
	RETURN;
END_IF

IF activeData.TcRelease() = 0 THEN
	activeData := 0;
END_IF

TryTcRelease := TRUE;
END_METHOD

END_FUNCTION_BLOCK

// Datatypes/Interfaces/Images/ITcVnImage/I_InterfaceDatatype_ITcVnImage
INTERFACE I_InterfaceDatatype_ITcVnImage EXTENDS I_InterfaceDatatype

PROPERTY PUBLIC Value : REFERENCE TO ITcVnImage
GET
END_GET
END_PROPERTY

END_INTERFACE

// Datatypes/Structs/_TcVnImageInfo
{attribute 'linkalways'} 
{attribute 'no_explicit_call' := 'This FB is a CLASS and must be accessed using methods or properties'}
{attribute 'enable_dynamic_creation'}
FUNCTION_BLOCK _TcVnImageInfo EXTENDS StructuredDatatypeBase
VAR
	localData : TcVnImageInfo;
	activeData : REFERENCE TO TcVnImageInfo REF= localData;
	_nImageSize : _ULINT(localData.nImageSize);
	_nWidth : _UDINT(localData.nWidth);
	_nHeight : _UDINT(localData.nHeight);
	_nXPadding : _UINT(localData.nXPadding);
	_nYPadding : _UINT(localData.nYPadding);
	_stPixelFormat : _TcVnPixelFormat();
END_VAR

PROPERTY PUBLIC Address : PVOID
GET
Address := ADR(activeData);
END_GET
END_PROPERTY

METHOD PUBLIC ClearReference
VAR_INPUT
END_VAR
activeData REF= localData;
SetMemberReference();
END_METHOD

PROPERTY PUBLIC Size : UDINT
GET
Size := SIZEOF(activeData);
END_GET
END_PROPERTY

METHOD FB_init : BOOL
VAR_INPUT
	bInitRetains : BOOL; // if TRUE, the retain variables are initialized (warm start / cold start)
	bInCopyCode : BOOL;  // if TRUE, the instance afterwards gets moved into the copy code (online change)
END_VAR
SetMemberReference();
AddMember('nImageSize',_nImageSize);
AddMember('nWidth',_nWidth);
AddMember('nHeight',_nHeight);
AddMember('nXPadding',_nXPadding);
AddMember('nYPadding',_nYPadding);
AddMember('stPixelFormat',_stPixelFormat);
END_METHOD

METHOD PROTECTED SetMemberReference
VAR_INPUT
END_VAR
_nImageSize.MakeReferenceTo(activeData.nImageSize);
_nWidth.MakeReferenceTo(activeData.nWidth);
_nHeight.MakeReferenceTo(activeData.nHeight);
_nXPadding.MakeReferenceTo(activeData.nXPadding);
_nYPadding.MakeReferenceTo(activeData.nYPadding);
_stPixelFormat.MakeReferenceTo(activeData.stPixelFormat);
END_METHOD

METHOD PUBLIC Clone : I_Datatype
VAR
    pClone : POINTER TO _TcVnImageInfo;
END_VAR
pClone := __NEW(_TcVnImageInfo());
pClone^.Value := Value;
Clone := pClone^;
END_METHOD

PROPERTY PUBLIC Identifier : T_MAXSTRING
GET
Identifier := 'TcVnImageInfo';
END_GET
END_PROPERTY

METHOD PUBLIC MakeReferenceTo
VAR_INPUT
	ReferenceTarget : REFERENCE TO TcVnImageInfo;
END_VAR
activeData REF= ReferenceTarget;
SetMemberReference();
END_METHOD

METHOD TryMakeReferenceTo : BOOL
VAR_INPUT
	Target : I_Datatype;
END_VAR
VAR
	pTargetData : POINTER TO TcVnImageInfo;
END_VAR
IF NOT IsEquivalentTo(Target) THEN
	RETURN;
END_IF

pTargetData := Target.Address;
activeData REF= pTargetData^;
SetMemberReference();
TryMakeReferenceTo := TRUE;
END_METHOD

PROPERTY PUBLIC Value : reference to TcVnImageInfo
GET
Value ref= activeData;
END_GET
END_PROPERTY

PROPERTY PUBLIC nHeight : Reference to _UDINT
GET
nHeight REF= _nHeight;
END_GET
END_PROPERTY

PROPERTY PUBLIC nImageSize : Reference to _ULINT
GET
nImageSize REF= _nImageSize;
END_GET
END_PROPERTY

PROPERTY PUBLIC nWidth : Reference to _UDINT
GET
nWidth REF= _nWidth;
END_GET
END_PROPERTY

PROPERTY PUBLIC nXPadding : Reference to _UINT
GET
nXPadding REF= _nXPadding;
END_GET
END_PROPERTY

PROPERTY PUBLIC nYPadding : Reference to _UINT
GET
nYPadding REF= _nYPadding;
END_GET
END_PROPERTY

PROPERTY PUBLIC stPixelFormat : Reference to _TcVnPixelFormat
GET
stPixelFormat REF= _stPixelFormat;
END_GET
END_PROPERTY

END_FUNCTION_BLOCK

// Datatypes/Structs/_TcVnPixelFormat
{attribute 'linkalways'} 
{attribute 'no_explicit_call' := 'This FB is a CLASS and must be accessed using methods or properties'}
{attribute 'enable_dynamic_creation'}
FUNCTION_BLOCK _TcVnPixelFormat EXTENDS StructuredDatatypeBase
VAR
	localData : TcVnPixelFormat;
	activeData : REFERENCE TO TcVnPixelFormat REF= localData;

	_bSupported : _BIT();
	_bSigned : _BIT();
	_bPlanar : _BIT();
	_bFloat : _BIT();
	_nChannels : _BYTE(localData.nChannels);
	_ePixelEncoding : _ETcVnPixelEncoding(localData.ePixelEncoding);
	_ePixelPackMode : _ETcVnPixelPackMode(localData.ePixelPackMode);
	_nElementSize : _UINT(localData.nElementSize);
	_nTotalSize : _UINT(localData.nTotalSize);
END_VAR

PROPERTY PUBLIC Address : PVOID
GET
Address := ADR(activeData);
END_GET
END_PROPERTY

METHOD PUBLIC ClearReference
VAR_INPUT
END_VAR
activeData REF= localData;
SetMemberReference();
END_METHOD

PROPERTY PUBLIC Size : UDINT
GET
Size := SIZEOF(activeData);
END_GET
END_PROPERTY

METHOD FB_init : BOOL
VAR_INPUT
	bInitRetains : BOOL; // if TRUE, the retain variables are initialized (warm start / cold start)
	bInCopyCode : BOOL;  // if TRUE, the instance afterwards gets moved into the copy code (online change)
END_VAR
SetMemberReference();
AddMember('bSupported',_bSupported);
AddMember('bSigned',_bSigned);
AddMember('bPlanar',_bPlanar);
AddMember('bFloat',_bFloat);
AddMember('nChannels',_nChannels);
AddMember('ePixelEncoding',_ePixelEncoding);
AddMember('ePixelPackMode',_ePixelPackMode);
AddMember('nElementSize',_nElementSize);
AddMember('nTotalSize',_nTotalSize);
END_METHOD

METHOD PROTECTED SetMemberReference
VAR_STAT
	// this variable is used for BITADR as this function fails if used on a local variable.
	structure : TcVnPixelFormat;
END_VAR
_bSupported.MakeReferenceTo(THIS^, GetByteOffset(localData, localData.bSupported), BITADR(structure.bSupported));
_bSigned.MakeReferenceTo(THIS^, GetByteOffset(localData, localData.bSigned), BITADR(structure.bSigned));
_bPlanar.MakeReferenceTo(THIS^, GetByteOffset(localData, localData.bPlanar), BITADR(structure.bPlanar));
_bFloat.MakeReferenceTo(THIS^, GetByteOffset(localData, localData.bFloat), BITADR(structure.bFloat));
_nChannels.MakeReferenceTo(activeData.nChannels);
_ePixelEncoding.MakeReferenceTo(activeData.ePixelEncoding);
_ePixelPackMode.MakeReferenceTo(activeData.ePixelPackMode);
_nElementSize.MakeReferenceTo(activeData.nElementSize);
_nTotalSize.MakeReferenceTo(activeData.nTotalSize);
END_METHOD

METHOD PUBLIC Clone : I_Datatype
VAR
    pClone : POINTER TO _TcVnPixelFormat;
END_VAR
pClone := __NEW(_TcVnPixelFormat());
pClone^.Value := Value;
Clone := pClone^;
END_METHOD

PROPERTY PUBLIC Identifier : T_MAXSTRING
GET
Identifier := 'TcVnPixelFormat';
END_GET
END_PROPERTY

METHOD PUBLIC MakeReferenceTo
VAR_INPUT
	ReferenceTarget : REFERENCE TO TcVnPixelFormat;
END_VAR
activeData REF= ReferenceTarget;
SetMemberReference();
END_METHOD

METHOD TryMakeReferenceTo : BOOL
VAR_INPUT
	Target : I_Datatype;
END_VAR
VAR
	pTargetData : POINTER TO TcVnPixelFormat;
END_VAR
IF NOT IsEquivalentTo(Target) THEN
	RETURN;
END_IF

pTargetData := Target.Address;
activeData REF= pTargetData^;
SetMemberReference();
TryMakeReferenceTo := TRUE;
END_METHOD

PROPERTY PUBLIC Value : reference to TcVnPixelFormat
GET
Value REF= activeData;
END_GET
END_PROPERTY

PROPERTY PUBLIC bFloat : Reference to _BIT
GET
bFloat REF= _bFloat;
END_GET
END_PROPERTY

PROPERTY PUBLIC bPlanar : Reference to _BIT
GET
bPlanar REF= _bPlanar;
END_GET
END_PROPERTY

PROPERTY PUBLIC bSigned : Reference to _BIT
GET
bSigned REF= _bSigned;
END_GET
END_PROPERTY

PROPERTY PUBLIC bSupported : Reference to _BIT
GET
bSupported REF= _bSupported;
END_GET
END_PROPERTY

PROPERTY PUBLIC ePixelEncoding : Reference to _ETcVnPixelEncoding
GET
ePixelEncoding REF= _ePixelEncoding;
END_GET
END_PROPERTY

PROPERTY PUBLIC ePixelPackMode : Reference to _ETcVnPixelPackMode
GET
ePixelPackMode REF= _ePixelPackMode;
END_GET
END_PROPERTY

PROPERTY PUBLIC nChannels : Reference to _BYTE
GET
nChannels REF= _nChannels;
END_GET
END_PROPERTY

PROPERTY PUBLIC nElementSize : Reference to _UINT
GET
nElementSize REF= _nElementSize;
END_GET
END_PROPERTY

PROPERTY PUBLIC nTotalSize : Reference to _UINT
GET
nTotalSize REF= _nTotalSize;
END_GET
END_PROPERTY

END_FUNCTION_BLOCK

// Datatypes/Enums/_ETcVnPixelEncoding
{attribute 'linkalways'} 
{attribute 'no_explicit_call' := 'This FB is a CLASS and must be accessed using methods or properties'}
{attribute 'enable_dynamic_creation'}
FUNCTION_BLOCK _ETcVnPixelEncoding EXTENDS EnumDatatypeBase
VAR
	localData : ETcVnPixelEncoding;
	activeData : REFERENCE TO ETcVnPixelEncoding;
	enumBaseDatatype : _BYTE(localData);
END_VAR

METHOD PROTECTED SetBaseDatatypeReference
VAR_INPUT
END_VAR
enumBaseDatatype.MakeReferenceTo(activeData);
END_METHOD

PROPERTY PUBLIC Address : PVOID
GET
Address := ADR(activeData);
END_GET
END_PROPERTY

METHOD PUBLIC ClearReference
VAR_INPUT
END_VAR
activeData REF= localData;
SetBaseDatatypeReference();
END_METHOD

PROPERTY PUBLIC Size : UDINT
GET
Size := SIZEOF(activeData);
END_GET
END_PROPERTY

METHOD FB_init : BOOL
VAR_INPUT
	bInitRetains : BOOL; // if TRUE, the retain variables are initialized (warm start / cold start)
	bInCopyCode : BOOL;  // if TRUE, the instance afterwards gets moved into the copy code (online change)
	InitialValue : ETcVnPixelEncoding;
END_VAR
localData := InitialValue;
AddBaseDatatype(enumBaseDatatype);
ClearReference();

AddLocalEnumeration('TCVN_PE_NONE', ETcVnPixelEncoding.TCVN_PE_NONE);
AddLocalEnumeration('TCVN_PE_BAYER_GR', ETcVnPixelEncoding.TCVN_PE_BAYER_GR);
AddLocalEnumeration('TCVN_PE_BAYER_RG', ETcVnPixelEncoding.TCVN_PE_BAYER_RG);
AddLocalEnumeration('TCVN_PE_BAYER_GB', ETcVnPixelEncoding.TCVN_PE_BAYER_GB);
AddLocalEnumeration('TCVN_PE_BAYER_BG', ETcVnPixelEncoding.TCVN_PE_BAYER_BG);
AddLocalEnumeration('TCVN_PE_YUV_411_UYYVYY', ETcVnPixelEncoding.TCVN_PE_YUV_411_UYYVYY);
AddLocalEnumeration('TCVN_PE_YUV_422_UYVY', ETcVnPixelEncoding.TCVN_PE_YUV_422_UYVY);
AddLocalEnumeration('TCVN_PE_YUV_422_YUYV', ETcVnPixelEncoding.TCVN_PE_YUV_422_YUYV);
AddLocalEnumeration('TCVN_PE_YCBCR_411_CBYYCRYY', ETcVnPixelEncoding.TCVN_PE_YCBCR_411_CBYYCRYY);
AddLocalEnumeration('TCVN_PE_YCBCR_422_CBYCRY', ETcVnPixelEncoding.TCVN_PE_YCBCR_422_CBYCRY);
AddLocalEnumeration('TCVN_PE_YCBCR_422_YCBYCR', ETcVnPixelEncoding.TCVN_PE_YCBCR_422_YCBYCR);
END_METHOD

METHOD PRIVATE AddLocalEnumeration
VAR_INPUT
	Enumeration : T_MAXSTRING;
	Value : ETcVnPixelEncoding;
END_VAR
AddEnumeration(Enumeration, Value);
END_METHOD

METHOD IsEnumeratorValueEqual : BOOL
VAR_INPUT
	Enumerator : I_KeyValueForwardEnumerator;
END_VAR
VAR
	storedValue : ETcVnPixelEncoding;
END_VAR
IF NOT Enumerator.TryGet(storedValue) THEN
	RETURN;
END_IF

IsEnumeratorValueEqual := storedValue = activeData;
END_METHOD

METHOD PUBLIC Clone : I_Datatype
VAR
    pClone : POINTER TO _ETcVnPixelEncoding;
END_VAR
pClone := __NEW(_ETcVnPixelEncoding(InitialValue := Value));
Clone := pClone^;
END_METHOD

PROPERTY PUBLIC Identifier : T_MAXSTRING
GET
Identifier := 'ETcVnPixelEncoding';
END_GET
END_PROPERTY

METHOD PUBLIC MakeReferenceTo
VAR_INPUT
	ReferenceTarget : REFERENCE TO ETcVnPixelEncoding;
END_VAR
activeData REF= ReferenceTarget;
SetBaseDatatypeReference();
END_METHOD

METHOD TryMakeReferenceTo : BOOL
VAR_INPUT
	Target : I_Datatype;
END_VAR
VAR
	pTargetData : POINTER TO ETcVnPixelEncoding;
END_VAR
IF NOT IsEquivalentTo(Target) THEN
	RETURN;
END_IF

pTargetData := Target.Address;
activeData REF= pTargetData^;
SetBaseDatatypeReference();
TryMakeReferenceTo := TRUE;
END_METHOD

PROPERTY PUBLIC Value : ETcVnPixelEncoding
GET
Value := activeData;
END_GET
SET
activeData := Value;
END_SET
END_PROPERTY

END_FUNCTION_BLOCK

// Datatypes/Enums/_ETcVnPixelPackMode
{attribute 'linkalways'} 
{attribute 'no_explicit_call' := 'This FB is a CLASS and must be accessed using methods or properties'}
{attribute 'enable_dynamic_creation'}
FUNCTION_BLOCK _ETcVnPixelPackMode EXTENDS EnumDatatypeBase
VAR
	localData : ETcVnPixelPackMode;
	activeData : REFERENCE TO ETcVnPixelPackMode;
	enumBaseDatatype : _BYTE(localData);
END_VAR

METHOD PROTECTED SetBaseDatatypeReference
VAR_INPUT
END_VAR
enumBaseDatatype.MakeReferenceTo(activeData);
END_METHOD

PROPERTY PUBLIC Address : PVOID
GET
Address := ADR(activeData);
END_GET
END_PROPERTY

METHOD PUBLIC ClearReference
VAR_INPUT
END_VAR
activeData REF= localData;
SetBaseDatatypeReference();
END_METHOD

PROPERTY PUBLIC Size : UDINT
GET
Size := SIZEOF(activeData);
END_GET
END_PROPERTY

METHOD FB_init : BOOL
VAR_INPUT
	bInitRetains : BOOL; // if TRUE, the retain variables are initialized (warm start / cold start)
	bInCopyCode : BOOL;  // if TRUE, the instance afterwards gets moved into the copy code (online change)
	InitialValue : ETcVnPixelPackMode;
END_VAR
localData := InitialValue;
AddBaseDatatype(enumBaseDatatype);
ClearReference();

AddLocalEnumeration('TCVN_PPM_NONE', ETcVnPixelPackMode.TCVN_PPM_NONE);
AddLocalEnumeration('TCVN_PPM_MONO1P', ETcVnPixelPackMode.TCVN_PPM_MONO1P);
AddLocalEnumeration('TCVN_PPM_MONO2P', ETcVnPixelPackMode.TCVN_PPM_MONO2P);
AddLocalEnumeration('TCVN_PPM_MONO4P', ETcVnPixelPackMode.TCVN_PPM_MONO4P);
AddLocalEnumeration('TCVN_PPM_MONO10PACKED', ETcVnPixelPackMode.TCVN_PPM_MONO10PACKED);
AddLocalEnumeration('TCVN_PPM_MONO12PACKED', ETcVnPixelPackMode.TCVN_PPM_MONO12PACKED);
AddLocalEnumeration('TCVN_PPM_RGB10V1PACKED', ETcVnPixelPackMode.TCVN_PPM_RGB10V1PACKED);
AddLocalEnumeration('TCVN_PPM_RGB10P32', ETcVnPixelPackMode.TCVN_PPM_RGB10P32);
AddLocalEnumeration('TCVN_PPM_RGB12V1PACKED', ETcVnPixelPackMode.TCVN_PPM_RGB12V1PACKED);
AddLocalEnumeration('TCVN_PPM_RGB565P', ETcVnPixelPackMode.TCVN_PPM_RGB565P);
AddLocalEnumeration('TCVN_PPM_BGR565P', ETcVnPixelPackMode.TCVN_PPM_BGR565P);
AddLocalEnumeration('TCVN_PPM_MONO10P', ETcVnPixelPackMode.TCVN_PPM_MONO10P);
AddLocalEnumeration('TCVN_PPM_MONO12P', ETcVnPixelPackMode.TCVN_PPM_MONO12P);
// AddLocalEnumeration('TCVN_PPM_MONO14P', ETcVnPixelPackMode.TCVN_PPM_MONO14P);
END_METHOD

METHOD PRIVATE AddLocalEnumeration
VAR_INPUT
	Enumeration : T_MAXSTRING;
	Value : ETcVnPixelPackMode;
END_VAR
AddEnumeration(Enumeration, Value);
END_METHOD

METHOD IsEnumeratorValueEqual : BOOL
VAR_INPUT
	Enumerator : I_KeyValueForwardEnumerator;
END_VAR
VAR
	storedValue : ETcVnPixelPackMode;
END_VAR
IF NOT Enumerator.TryGet(storedValue) THEN
	RETURN;
END_IF

IsEnumeratorValueEqual := storedValue = activeData;
END_METHOD

METHOD PUBLIC Clone : I_Datatype
VAR
    pClone : POINTER TO _ETcVnPixelPackMode;
END_VAR
pClone := __NEW(_ETcVnPixelPackMode(InitialValue := Value));
Clone := pClone^;
END_METHOD

PROPERTY PUBLIC Identifier : T_MAXSTRING
GET
Identifier := 'ETcVnPixelPackMode';
END_GET
END_PROPERTY

METHOD PUBLIC MakeReferenceTo
VAR_INPUT
	ReferenceTarget : REFERENCE TO ETcVnPixelPackMode;
END_VAR
activeData REF= ReferenceTarget;
SetBaseDatatypeReference();
END_METHOD

METHOD TryMakeReferenceTo : BOOL
VAR_INPUT
	Target : I_Datatype;
END_VAR
VAR
	pTargetData : POINTER TO ETcVnPixelPackMode;
END_VAR
IF NOT IsEquivalentTo(Target) THEN
	RETURN;
END_IF

pTargetData := Target.Address;
activeData REF= pTargetData^;
SetBaseDatatypeReference();
TryMakeReferenceTo := TRUE;
END_METHOD

PROPERTY PUBLIC Value : ETcVnPixelPackMode
GET
Value := activeData;
END_GET
SET
activeData := Value;
END_SET
END_PROPERTY

END_FUNCTION_BLOCK

// Datatypes/Aliases/_TcVnArray3_Point2_REAL
{attribute 'linkalways'} 
{attribute 'no_explicit_call' := 'This FB is a CLASS and must be accessed using methods or properties'}
{attribute 'enable_dynamic_creation'}
FUNCTION_BLOCK _TcVnArray3_Point2_REAL EXTENDS AliasDatatypeBase
VAR
	localData : TcVnArray3_Point2_REAL;
	activeData : REFERENCE TO TcVnArray3_Point2_REAL REF= localData;
	aliasBaseDatatype : _Array0to2OfTcVnPoint2_REAL;
END_VAR

METHOD PROTECTED SetBaseDatatypeReference
VAR_INPUT
END_VAR
aliasBaseDatatype.MakeReferenceTo(activeData);
END_METHOD

PROPERTY PUBLIC Address : PVOID
GET
Address := ADR(activeData);
END_GET
END_PROPERTY

METHOD PUBLIC ClearReference
VAR_INPUT
END_VAR
activeData REF= localData;
SetBaseDatatypeReference();
END_METHOD

PROPERTY PUBLIC Size : UDINT
GET
Size := SIZEOF(activeData);
END_GET
END_PROPERTY

METHOD FB_init : BOOL
VAR_INPUT
	bInitRetains : BOOL; // if TRUE, the retain variables are initialized (warm start / cold start)
	bInCopyCode : BOOL;  // if TRUE, the instance afterwards gets moved into the copy code (online change)
	//InitialValue : TcVnArray4_LREAL; // if possible, not all values can be initialized
END_VAR
//localData := InitialValue; // if possible, not all values can be initialized
SetBaseDatatypeReference();
AddBaseDatatype(aliasBaseDatatype);
END_METHOD

METHOD PUBLIC Clone : I_Datatype
VAR
    pClone : POINTER TO _TcVnArray3_Point2_REAL;
END_VAR
pClone := __NEW(_TcVnArray3_Point2_REAL);
Clone := pClone^;
END_METHOD

PROPERTY PUBLIC Identifier : T_MAXSTRING
GET
Identifier := 'TcVnArray3_Point2_REAL';
END_GET
END_PROPERTY

METHOD PUBLIC MakeReferenceTo
VAR_INPUT
	ReferenceTarget : REFERENCE TO TcVnArray3_Point2_REAL;
END_VAR
activeData REF= ReferenceTarget;
SetBaseDatatypeReference();
END_METHOD

METHOD TryMakeReferenceTo : BOOL
VAR_INPUT
	Target : I_Datatype;
END_VAR
VAR
	pTargetData : POINTER TO TcVnArray3_Point2_REAL;
END_VAR
IF NOT IsEquivalentTo(Target) THEN
	RETURN;
END_IF

pTargetData := Target.Address;
activeData REF= pTargetData^;
SetBaseDatatypeReference();
TryMakeReferenceTo := TRUE;
END_METHOD

PROPERTY PUBLIC Value : REFERENCE TO TcVnArray3_Point2_REAL
GET
Value REF= activeData;
END_GET
END_PROPERTY

END_FUNCTION_BLOCK

// Datatypes/Arrays/_Array0to2OfTcVnPoint2_REAL
{attribute 'linkalways'} 
{attribute 'no_explicit_call' := 'This FB is a CLASS and must be accessed using methods or properties'}
{attribute 'enable_dynamic_creation'}
FUNCTION_BLOCK _Array0to2OfTcVnPoint2_REAL EXTENDS ArrayDatatypeBase_1D
VAR CONSTANT
	lBound : DINT := 0;
	uBound : DINT := 2;
END_VAR
VAR
	localData : ARRAY [lBound..uBound] OF TcVnPoint2_REAL;
	activeData : REFERENCE TO ARRAY [lBound..uBound] OF TcVnPoint2_REAL REF= localData;
	elements : ARRAY [lBound..uBound] OF _TcVnPoint2_REAL;
	baseType : _TcVnPoint2_REAL;
END_VAR

METHOD FB_init : BOOL
VAR_INPUT
	bInitRetains : BOOL; // if TRUE, the retain variables are initialized (warm start / cold start)
	bInCopyCode : BOOL;  // if TRUE, the instance afterwards gets moved into the copy code (online change)
END_VAR
SetElementReference();
END_METHOD

METHOD PROTECTED OnSerializeArrayValues
VAR_INPUT
	Serializer : I_Serializer;
END_VAR
VAR
	i : DINT;
END_VAR
FOR i := lBound TO uBound DO
	elements[i].SerializeWith(Serializer);
END_FOR
END_METHOD

METHOD PROTECTED SetElementReference
VAR_INPUT
END_VAR
VAR
	i : DINT;
END_VAR
FOR i := lBound TO uBound DO
	elements[i].MakeReferenceTo(activeData[i]);
END_FOR
END_METHOD

METHOD PROTECTED TryDeserializeArrayValues : BOOL
VAR_INPUT
	Deserializer : I_Deserializer;
	Feedback : I_DeserializerFeedback;
END_VAR
VAR
	enumerator : I_DeserializerArrayForwardEnumerator;
	i : DINT;
END_VAR
enumerator := Deserializer.GetArrayEnumerator();
i := lBound;

WHILE enumerator.MoveNext() AND i <= uBound DO
	
	IF NOT elements[i].TryDeserializeFrom(enumerator.Current, Feedback) THEN
		EXIT;
	END_IF
	i := i + 1;

END_WHILE
enumerator.Dispose();
END_METHOD

PROPERTY PUBLIC Address : PVOID
GET
Address := ADR(activeData);
END_GET
END_PROPERTY

PROPERTY PUBLIC BaseDatatype : I_Datatype
GET
BaseDatatype := baseType;
END_GET
END_PROPERTY

METHOD PUBLIC ClearReference
VAR_INPUT
END_VAR
activeData REF= localData;
SetElementReference();
END_METHOD

PROPERTY PUBLIC Size : UDINT
GET
Size := SIZEOF(activeData);
END_GET
END_PROPERTY

METHOD PUBLIC TryGetElementAsDatatypeByIndex : BOOL
VAR_INPUT
	Index : DINT;
	Destination : REFERENCE TO I_Datatype;
END_VAR
IF Index < lbound OR Index > ubound THEN
	RETURN;
END_IF

Destination := elements[Index];
TryGetElementAsDatatypeByIndex := TRUE;
END_METHOD

METHOD PUBLIC TryGetLowerBound : BOOL
VAR_INPUT
	Dimention : UDINT;
	Destination : REFERENCE TO DINT;
END_VAR
IF Dimention = 1 THEN
	Destination := lBound;
	TryGetLowerBound := TRUE;
END_IF
END_METHOD

METHOD PUBLIC TryGetUpperBound : BOOL
VAR_INPUT
	Dimention : UDINT;
	Destination : REFERENCE TO DINT;
END_VAR
IF Dimention = 1 THEN
	Destination := uBound;
	TryGetUpperBound := TRUE;
END_IF
END_METHOD

METHOD PUBLIC Clone : I_Datatype
VAR
    pClone : POINTER TO _Array0to2OfTcVnPoint2_REAL;
END_VAR
pClone := __NEW(_Array0to2OfTcVnPoint2_REAL());
pClone^.Value := Value;
Clone := pClone^;
END_METHOD

METHOD PUBLIC MakeReferenceTo
VAR_INPUT
	ReferenceTarget : REFERENCE TO ARRAY [lBound..uBound] OF TcVnPoint2_REAL;
END_VAR
activeData REF= ReferenceTarget;
SetElementReference();
END_METHOD

METHOD TryMakeReferenceTo : BOOL
VAR_INPUT
	Target : I_Datatype;
END_VAR
VAR
	pTargetData : POINTER TO ARRAY [lBound..uBound] OF TcVnPoint2_REAL;
END_VAR
IF NOT IsEquivalentTo(Target) THEN
	RETURN;
END_IF

pTargetData := Target.Address;
activeData REF= pTargetData^;
SetElementReference();
TryMakeReferenceTo := TRUE;
END_METHOD

PROPERTY PUBLIC Value : REFERENCE TO ARRAY [lBound..uBound] OF TcVnPoint2_REAL;
GET
Value ref= activeData;
END_GET
END_PROPERTY

END_FUNCTION_BLOCK

// Datatypes/Aliases/_TcVnPoint2_REAL
{attribute 'linkalways'} 
{attribute 'no_explicit_call' := 'This FB is a CLASS and must be accessed using methods or properties'}
{attribute 'enable_dynamic_creation'}
FUNCTION_BLOCK _TcVnPoint2_REAL EXTENDS AliasDatatypeBase
VAR
	localData : TcVnPoint2_REAL;
	activeData : REFERENCE TO TcVnPoint2_REAL REF= localData;
	aliasBaseDatatype : _TcVnVector2_REAL;
END_VAR

METHOD PROTECTED SetBaseDatatypeReference
VAR_INPUT
END_VAR
aliasBaseDatatype.MakeReferenceTo(activeData);
END_METHOD

PROPERTY PUBLIC Address : PVOID
GET
Address := ADR(activeData);
END_GET
END_PROPERTY

METHOD PUBLIC ClearReference
VAR_INPUT
END_VAR
activeData REF= localData;
SetBaseDatatypeReference();
END_METHOD

PROPERTY PUBLIC Size : UDINT
GET
Size := SIZEOF(activeData);
END_GET
END_PROPERTY

METHOD FB_init : BOOL
VAR_INPUT
	bInitRetains : BOOL; // if TRUE, the retain variables are initialized (warm start / cold start)
	bInCopyCode : BOOL;  // if TRUE, the instance afterwards gets moved into the copy code (online change)
	//InitialValue : <type>; // if possible, not all values can be initialized
END_VAR
//localData := InitialValue; // if possible, not all values can be initialized
SetBaseDatatypeReference();
AddBaseDatatype(aliasBaseDatatype);
END_METHOD

METHOD PUBLIC Clone : I_Datatype
VAR
    pClone : POINTER TO _TcVnPoint2_REAL;
END_VAR
pClone := __NEW(_TcVnPoint2_REAL);
Clone := pClone^;
END_METHOD

PROPERTY PUBLIC Identifier : T_MAXSTRING
GET
Identifier := 'TcVnPoint2_REAL';
END_GET
END_PROPERTY

METHOD PUBLIC MakeReferenceTo
VAR_INPUT
	ReferenceTarget : REFERENCE TO TcVnPoint2_REAL;
END_VAR
activeData REF= ReferenceTarget;
SetBaseDatatypeReference();
END_METHOD

METHOD TryMakeReferenceTo : BOOL
VAR_INPUT
	Target : I_Datatype;
END_VAR
VAR
	pTargetData : POINTER TO TcVnPoint2_REAL;
END_VAR
IF NOT IsEquivalentTo(Target) THEN
	RETURN;
END_IF

pTargetData := Target.Address;
activeData REF= pTargetData^;
SetBaseDatatypeReference();
TryMakeReferenceTo := TRUE;
END_METHOD

PROPERTY PUBLIC Value : REFERENCE TO TcVnPoint2_REAL
GET
Value REF= activeData;
END_GET
END_PROPERTY

END_FUNCTION_BLOCK

// Datatypes/Aliases/_TcVnVector2_REAL
{attribute 'linkalways'} 
{attribute 'no_explicit_call' := 'This FB is a CLASS and must be accessed using methods or properties'}
{attribute 'enable_dynamic_creation'}
FUNCTION_BLOCK _TcVnVector2_REAL EXTENDS AliasDatatypeBase
VAR
	localData : TcVnVector2_REAL;
	activeData : REFERENCE TO TcVnVector2_REAL REF= localData;
	aliasBaseDatatype : _Array0to1OfREAL;
END_VAR

METHOD PROTECTED SetBaseDatatypeReference
VAR_INPUT
END_VAR
aliasBaseDatatype.MakeReferenceTo(activeData);
END_METHOD

PROPERTY PUBLIC Address : PVOID
GET
Address := ADR(activeData);
END_GET
END_PROPERTY

METHOD PUBLIC ClearReference
VAR_INPUT
END_VAR
activeData REF= localData;
SetBaseDatatypeReference();
END_METHOD

PROPERTY PUBLIC Size : UDINT
GET
Size := SIZEOF(activeData);
END_GET
END_PROPERTY

METHOD FB_init : BOOL
VAR_INPUT
	bInitRetains : BOOL; // if TRUE, the retain variables are initialized (warm start / cold start)
	bInCopyCode : BOOL;  // if TRUE, the instance afterwards gets moved into the copy code (online change)
	//InitialValue : <type>; // if possible, not all values can be initialized
END_VAR
//localData := InitialValue; // if possible, not all values can be initialized
SetBaseDatatypeReference();
AddBaseDatatype(aliasBaseDatatype);
END_METHOD

METHOD PUBLIC Clone : I_Datatype
VAR
    pClone : POINTER TO _TcVnVector2_REAL;
END_VAR
pClone := __NEW(_TcVnVector2_REAL);
Clone := pClone^;
END_METHOD

PROPERTY PUBLIC Identifier : T_MAXSTRING
GET
Identifier := 'TcVnVector2_REAL';
END_GET
END_PROPERTY

METHOD PUBLIC MakeReferenceTo
VAR_INPUT
	ReferenceTarget : REFERENCE TO TcVnVector2_REAL;
END_VAR
activeData REF= ReferenceTarget;
SetBaseDatatypeReference();
END_METHOD

METHOD TryMakeReferenceTo : BOOL
VAR_INPUT
	Target : I_Datatype;
END_VAR
VAR
	pTargetData : POINTER TO TcVnVector2_REAL;
END_VAR
IF NOT IsEquivalentTo(Target) THEN
	RETURN;
END_IF

pTargetData := Target.Address;
activeData REF= pTargetData^;
SetBaseDatatypeReference();
TryMakeReferenceTo := TRUE;
END_METHOD

PROPERTY PUBLIC Value : REFERENCE TO TcVnVector2_REAL
GET
Value REF= activeData;
END_GET
END_PROPERTY

END_FUNCTION_BLOCK

// Datatypes/Arrays/_Array0to1OfREAL
{attribute 'linkalways'} 
{attribute 'no_explicit_call' := 'This FB is a CLASS and must be accessed using methods or properties'}
{attribute 'enable_dynamic_creation'}
FUNCTION_BLOCK _Array0to1OfREAL EXTENDS ArrayDatatypeBase_1D
VAR CONSTANT
	lBound : DINT := 0;
	uBound : DINT := 1;
END_VAR
VAR
	localData : ARRAY [lBound..uBound] OF REAL;
	activeData : REFERENCE TO ARRAY [lBound..uBound] OF REAL REF= localData;
	elements : ARRAY [lBound..uBound] OF _REAL(0.0);
	baseType : _REAL(0.0);
END_VAR

METHOD FB_init : BOOL
VAR_INPUT
	bInitRetains : BOOL; // if TRUE, the retain variables are initialized (warm start / cold start)
	bInCopyCode : BOOL;  // if TRUE, the instance afterwards gets moved into the copy code (online change)
END_VAR
SetElementReference();
END_METHOD

METHOD PROTECTED OnSerializeArrayValues
VAR_INPUT
	Serializer : I_Serializer;
END_VAR
VAR
	i : DINT;
END_VAR
FOR i := lBound TO uBound DO
	elements[i].SerializeWith(Serializer);
END_FOR
END_METHOD

METHOD PROTECTED SetElementReference
VAR_INPUT
END_VAR
VAR
	i : DINT;
END_VAR
FOR i := lBound TO uBound DO
	elements[i].MakeReferenceTo(activeData[i]);
END_FOR
END_METHOD

METHOD PROTECTED TryDeserializeArrayValues : BOOL
VAR_INPUT
	Deserializer : I_Deserializer;
	Feedback : I_DeserializerFeedback;
END_VAR
VAR
	enumerator : I_DeserializerArrayForwardEnumerator;
	i : DINT;
END_VAR
enumerator := Deserializer.GetArrayEnumerator();
i := lBound;

WHILE enumerator.MoveNext() AND i <= uBound DO
	
	IF NOT elements[i].TryDeserializeFrom(enumerator.Current, Feedback) THEN
		EXIT;
	END_IF
	i := i + 1;

END_WHILE
enumerator.Dispose();
END_METHOD

PROPERTY PUBLIC Address : PVOID
GET
Address := ADR(activeData);
END_GET
END_PROPERTY

PROPERTY PUBLIC BaseDatatype : I_Datatype
GET
BaseDatatype := baseType;
END_GET
END_PROPERTY

METHOD PUBLIC ClearReference
VAR_INPUT
END_VAR
activeData REF= localData;
SetElementReference();
END_METHOD

PROPERTY PUBLIC Size : UDINT
GET
Size := SIZEOF(activeData);
END_GET
END_PROPERTY

METHOD PUBLIC TryGetElementAsDatatypeByIndex : BOOL
VAR_INPUT
	Index : DINT;
	Destination : REFERENCE TO I_Datatype;
END_VAR
IF Index < lbound OR Index > ubound THEN
	RETURN;
END_IF

Destination := elements[Index];
TryGetElementAsDatatypeByIndex := TRUE;
END_METHOD

METHOD PUBLIC TryGetLowerBound : BOOL
VAR_INPUT
	Dimention : UDINT;
	Destination : REFERENCE TO DINT;
END_VAR
IF Dimention = 1 THEN
	Destination := lBound;
	TryGetLowerBound := TRUE;
END_IF
END_METHOD

METHOD PUBLIC TryGetUpperBound : BOOL
VAR_INPUT
	Dimention : UDINT;
	Destination : REFERENCE TO DINT;
END_VAR
IF Dimention = 1 THEN
	Destination := uBound;
	TryGetUpperBound := TRUE;
END_IF
END_METHOD

METHOD PUBLIC Clone : I_Datatype
VAR
    pClone : POINTER TO _Array0to1OfREAL;
END_VAR
pClone := __NEW(_Array0to1OfREAL());
pClone^.Value := Value;
Clone := pClone^;
END_METHOD

METHOD PUBLIC MakeReferenceTo
VAR_INPUT
	ReferenceTarget : REFERENCE TO ARRAY [lBound..uBound] OF REAL;
END_VAR
activeData REF= ReferenceTarget;
SetElementReference();
END_METHOD

METHOD TryMakeReferenceTo : BOOL
VAR_INPUT
	Target : I_Datatype;
END_VAR
VAR
	pTargetData : POINTER TO ARRAY [lBound..uBound] OF REAL;
END_VAR
IF NOT IsEquivalentTo(Target) THEN
	RETURN;
END_IF

pTargetData := Target.Address;
activeData REF= pTargetData^;
SetElementReference();
TryMakeReferenceTo := TRUE;
END_METHOD

PROPERTY PUBLIC Value : REFERENCE TO ARRAY [lBound..uBound] OF REAL;
GET
Value ref= activeData;
END_GET
END_PROPERTY

END_FUNCTION_BLOCK

